LIN {X 0,Y 406.191,Z 782.909,A -85,B 0,C 180,E1 -7084.724,E2 -7084.724} C_VEL
LIN {X 0,Y 404.548,Z 789.361,A -85,B 0,C 180,E1 -7085.289,E2 -7085.289} C_VEL
LIN {X 0,Y 396.99,Z 805.186,A -85,B 0,C 180,E1 -7086.699,E2 -7086.699} C_VEL
LIN {X 0,Y 395.215,Z 810.941,A -85,B 0,C 180,E1 -7087.406,E2 -7087.406} C_VEL
LIN {X 0,Y 393.105,Z 824.076,A -85,B 0,C 180,E1 -7089.452,E2 -7089.452} C_VEL
LIN {X 0,Y 391.138,Z 835.792,A -85,B 0,C 180,E1 -7091.674,E2 -7091.674} C_VEL
LIN {X 0,Y 389.418,Z 846.025,A -85,B 0,C 180,E1 -7094.054,E2 -7094.054} C_VEL
LIN {X 0,Y 388.003,Z 854.789,A -85,B 0,C 180,E1 -7096.59,E2 -7096.59} C_VEL
LIN {X 0,Y 386.881,Z 862.038,A -85,B 0,C 180,E1 -7099.276,E2 -7099.276} C_VEL
LIN {X 0,Y 386.108,Z 867.692,A -85,B 0,C 180,E1 -7102.112,E2 -7102.112} C_VEL
LIN {X 0,Y 385.668,Z 871.52,A -85,B 0,C 180,E1 -7104.943,E2 -7104.943} C_VEL
LIN {X 0,Y 385.436,Z 873.652,A -85,B 0,C 180,E1 -7107.77,E2 -7107.77} C_VEL
LIN {X 0,Y 385.386,Z 874.148,A -85,B 0,C 180,E1 -7110.595,E2 -7110.595} C_VEL
LIN {X 0,Y 385.508,Z 872.915,A -85,B 0,C 180,E1 -7113.569,E2 -7113.569} C_VEL
LIN {X 0,Y 385.826,Z 870.044,A -85,B 0,C 180,E1 -7116.398,E2 -7116.398} C_VEL
LIN {X 0,Y 386.363,Z 865.702,A -85,B 0,C 180,E1 -7119.083,E2 -7119.083} C_VEL
LIN {X 0,Y 387.229,Z 859.657,A -85,B 0,C 180,E1 -7121.771,E2 -7121.771} C_VEL
LIN {X 0,Y 388.409,Z 852.203,A -85,B 0,C 180,E1 -7124.308,E2 -7124.308} C_VEL
LIN {X 0,Y 389.961,Z 842.815,A -85,B 0,C 180,E1 -7126.842,E2 -7126.842} C_VEL
LIN {X 0,Y 391.848,Z 831.752,A -85,B 0,C 180,E1 -7129.245,E2 -7129.245} C_VEL
LIN {X 0,Y 393.914,Z 819.324,A -85,B 0,C 180,E1 -7131.439,E2 -7131.439} C_VEL
LIN {X 0,Y 396.073,Z 805.549,A -85,B 0,C 180,E1 -7133.429,E2 -7133.429} C_VEL
LIN {X 0,Y 398.217,Z 790.671,A -85,B 0,C 180,E1 -7135.188,E2 -7135.188} C_VEL
LIN {X 0,Y 400.199,Z 774.726,A -85,B 0,C 180,E1 -7136.726,E2 -7136.726} C_VEL
LIN {X 0,Y 401.902,Z 758.677,A -85,B 0,C 180,E1 -7137.971,E2 -7137.971} C_VEL
LIN {X 0,Y 403.321,Z 741.862,A -85,B 0,C 180,E1 -7139.001,E2 -7139.001} C_VEL
LIN {X 0,Y 404.378,Z 723.64,A -85,B 0,C 180,E1 -7139.842,E2 -7139.842} C_VEL
LIN {X 0,Y 404.994,Z 704.322,A -85,B 0,C 180,E1 -7140.452,E2 -7140.452} C_VEL
LIN {X 0,Y 406.775,Z 627.656,A -85,B 0,C 180,E1 -7141.895,E2 -7141.895} C_VEL
LIN {X 0,Y 409.987,Z 503.447,A -85,B 0,C 180,E1 -7144.179,E2 -7144.179} C_VEL
LIN {X 0,Y 409.147,Z 496.442,A -85,B 0,C 180,E1 -7144.454,E2 -7144.454} C_VEL
LIN {X 0,Y 410.584,Z 460.846,A -85,B 0,C 180,E1 -7147.153,E2 -7147.153} C_VEL
LIN {X 0,Y 411.5,Z 441.452,A -85,B 0,C 180,E1 -7148.742,E2 -7148.742} C_VEL
LIN {X 0,Y 404.352,Z 422.499,A -85,B 0,C 180,E1 -7151.318,E2 -7151.318} C_VEL
LIN {X 0,Y 399.341,Z 410.865,A -85,B 0,C 180,E1 -7153.021,E2 -7153.021} C_VEL
LIN {X 0,Y 398.731,Z 410.597,A -85,B 0,C 180,E1 -7153.158,E2 -7153.158} C_VEL
LIN {X 0,Y 405.761,Z 426.901,A -85,B 0,C 180,E1 -7156.118,E2 -7156.118} C_VEL
LIN {X 0,Y 412.622,Z 444.419,A -85,B 0,C 180,E1 -7159.01,E2 -7159.01} C_VEL
LIN {X 0,Y 414.278,Z 448.803,A -85,B 0,C 180,E1 -7159.7,E2 -7159.7} C_VEL
LIN {X 0,Y 409.876,Z 489.947,A -85,B 0,C 180,E1 -7163.645,E2 -7163.645} C_VEL
LIN {X 0,Y 405.47,Z 533.935,A -85,B 0,C 180,E1 -7167.816,E2 -7167.816} C_VEL
LIN {X 0,Y 401.479,Z 578.727,A -85,B 0,C 180,E1 -7172.001,E2 -7172.001} C_VEL
LIN {X 0,Y 399.443,Z 605.362,A -85,B 0,C 180,E1 -7174.432,E2 -7174.432} C_VEL
LIN {X 0,Y 400.173,Z 614.62,A -85,B 0,C 180,E1 -7174.744,E2 -7174.744} C_VEL
LIN {X 0,Y 394.659,Z 751.079,A -85,B 0,C 180,E1 -7178.197,E2 -7178.197} C_VEL
LIN {X 0,Y 394.114,Z 767.215,A -85,B 0,C 180,E1 -7178.833,E2 -7178.833} C_VEL
LIN {X 0,Y 393.253,Z 783.894,A -85,B 0,C 180,E1 -7179.77,E2 -7179.77} C_VEL
LIN {X 0,Y 392.264,Z 798.711,A -85,B 0,C 180,E1 -7180.88,E2 -7180.88} C_VEL
LIN {X 0,Y 391.095,Z 813.488,A -85,B 0,C 180,E1 -7182.288,E2 -7182.288} C_VEL
LIN {X 0,Y 389.952,Z 826.524,A -85,B 0,C 180,E1 -7183.847,E2 -7183.847} C_VEL
LIN {X 0,Y 388.794,Z 839.087,A -85,B 0,C 180,E1 -7185.706,E2 -7185.706} C_VEL
LIN {X 0,Y 387.824,Z 849.553,A -85,B 0,C 180,E1 -7187.644,E2 -7187.644} C_VEL
LIN {X 0,Y 386.992,Z 859.155,A -85,B 0,C 180,E1 -7189.862,E2 -7189.862} C_VEL
LIN {X 0,Y 386.402,Z 866.658,A -85,B 0,C 180,E1 -7192.117,E2 -7192.117} C_VEL
LIN {X 0,Y 386.036,Z 872.623,A -85,B 0,C 180,E1 -7194.5,E2 -7194.5} C_VEL
LIN {X 0,Y 385.892,Z 876.86,A -85,B 0,C 180,E1 -7197.029,E2 -7197.029} C_VEL
LIN {X 0,Y 385.925,Z 879.099,A -85,B 0,C 180,E1 -7199.406,E2 -7199.406} C_VEL
LIN {X 0,Y 386.147,Z 879.624,A -85,B 0,C 180,E1 -7201.929,E2 -7201.929} C_VEL
LIN {X 0,Y 386.531,Z 878.409,A -85,B 0,C 180,E1 -7204.302,E2 -7204.302} C_VEL
LIN {X 0,Y 387.2,Z 875.274,A -85,B 0,C 180,E1 -7206.822,E2 -7206.822} C_VEL
LIN {X 0,Y 388.11,Z 870.426,A -85,B 0,C 180,E1 -7209.191,E2 -7209.191} C_VEL
LIN {X 0,Y 389.28,Z 864.13,A -85,B 0,C 180,E1 -7211.406,E2 -7211.406} C_VEL
LIN {X 0,Y 390.71,Z 855.743,A -85,B 0,C 180,E1 -7213.617,E2 -7213.617} C_VEL
LIN {X 0,Y 392.242,Z 846.555,A -85,B 0,C 180,E1 -7215.524,E2 -7215.524} C_VEL
LIN {X 0,Y 394.103,Z 834.538,A -85,B 0,C 180,E1 -7217.496,E2 -7217.496} C_VEL
LIN {X 0,Y 395.961,Z 821.007,A -85,B 0,C 180,E1 -7219.24,E2 -7219.24} C_VEL
LIN {X 0,Y 397.722,Z 805.897,A -85,B 0,C 180,E1 -7220.76,E2 -7220.76} C_VEL
LIN {X 0,Y 399.098,Z 790.974,A -85,B 0,C 180,E1 -7221.918,E2 -7221.918} C_VEL
LIN {X 0,Y 400.201,Z 775.813,A -85,B 0,C 180,E1 -7222.822,E2 -7222.822} C_VEL
LIN {X 0,Y 402.733,Z 747.163,A -85,B 0,C 180,E1 -7224.182,E2 -7224.182} C_VEL
LIN {X 0,Y 414.664,Z 670.102,A -85,B 0,C 180,E1 -7227.461,E2 -7227.461} C_VEL
LIN {X 0,Y 419.144,Z 642.978,A -85,B 0,C 180,E1 -7228.495,E2 -7228.495} C_VEL
LIN {X 0,Y 425.346,Z 629.291,A -85,B 0,C 180,E1 -7229.425,E2 -7229.425} C_VEL
LIN {X 0,Y 433.429,Z 606.324,A -85,B 0,C 180,E1 -7232.2,E2 -7232.2} C_VEL
LIN {X 0,Y 442.63,Z 586.799,A -85,B 0,C 180,E1 -7234.697,E2 -7234.697} C_VEL
LIN {X 0,Y 451.342,Z 572.774,A -85,B 0,C 180,E1 -7236.588,E2 -7236.588} C_VEL
LIN {X 0,Y 449.087,Z 580.004,A -85,B 0,C 180,E1 -7238.239,E2 -7238.239} C_VEL
LIN {X 0,Y 449.02,Z 587.826,A -85,B 0,C 180,E1 -7240.003,E2 -7240.003} C_VEL
LIN {X 0,Y 451.418,Z 596.121,A -85,B 0,C 180,E1 -7241.812,E2 -7241.812} C_VEL
LIN {X 0,Y 456.495,Z 604.734,A -85,B 0,C 180,E1 -7243.625,E2 -7243.625} C_VEL
LIN {X 0,Y 459.602,Z 608.735,A -85,B 0,C 180,E1 -7244.43,E2 -7244.43} C_VEL
LIN {X 0,Y 448.07,Z 630.938,A -85,B 0,C 180,E1 -7244.977,E2 -7244.977} C_VEL
LIN {X 0,Y 439.647,Z 649.717,A -85,B 0,C 180,E1 -7245.626,E2 -7245.626} C_VEL
LIN {X 0,Y 428.488,Z 674.951,A -85,B 0,C 180,E1 -7246.527,E2 -7246.527} C_VEL
LIN {X 0,Y 420.017,Z 698.201,A -85,B 0,C 180,E1 -7247.552,E2 -7247.552} C_VEL
LIN {X 0,Y 416.651,Z 725.416,A -85,B 0,C 180,E1 -7248.015,E2 -7248.015} C_VEL
LIN {X 0,Y 414.363,Z 753.273,A -85,B 0,C 180,E1 -7248.807,E2 -7248.807} C_VEL
LIN {X 0,Y 411.564,Z 778.053,A -85,B 0,C 180,E1 -7249.742,E2 -7249.742} C_VEL
LIN {X 0,Y 408.571,Z 802.272,A -85,B 0,C 180,E1 -7250.938,E2 -7250.938} C_VEL
LIN {X 0,Y 405.472,Z 825.859,A -85,B 0,C 180,E1 -7252.387,E2 -7252.387} C_VEL
LIN {X 0,Y 402.205,Z 849.287,A -85,B 0,C 180,E1 -7254.157,E2 -7254.157} C_VEL
LIN {X 0,Y 399.157,Z 870.873,A -85,B 0,C 180,E1 -7256.105,E2 -7256.105} C_VEL
LIN {X 0,Y 396.34,Z 890.303,A -85,B 0,C 180,E1 -7258.18,E2 -7258.18} C_VEL
LIN {X 0,Y 393.688,Z 908.695,A -85,B 0,C 180,E1 -7260.481,E2 -7260.481} C_VEL
LIN {X 0,Y 391.243,Z 925.999,A -85,B 0,C 180,E1 -7263.023,E2 -7263.023} C_VEL
LIN {X 0,Y 389.144,Z 941.582,A -85,B 0,C 180,E1 -7265.726,E2 -7265.726} C_VEL
LIN {X 0,Y 387.348,Z 956.066,A -85,B 0,C 180,E1 -7268.723,E2 -7268.723} C_VEL
LIN {X 0,Y 386.035,Z 968.119,A -85,B 0,C 180,E1 -7271.735,E2 -7271.735} C_VEL
LIN {X 0,Y 385.139,Z 978.117,A -85,B 0,C 180,E1 -7274.799,E2 -7274.799} C_VEL
LIN {X 0,Y 384.644,Z 985.702,A -85,B 0,C 180,E1 -7277.692,E2 -7277.692} C_VEL
LIN {X 0,Y 384.372,Z 991.86,A -85,B 0,C 180,E1 -7280.718,E2 -7280.718} C_VEL
LIN {X 0,Y 384.304,Z 996.2,A -85,B 0,C 180,E1 -7283.726,E2 -7283.726} C_VEL
LIN {X 0,Y 384.277,Z 998.794,A -85,B 0,C 180,E1 -7286.569,E2 -7286.569} C_VEL
LIN {X 0,Y 384.268,Z 999.915,A -85,B 0,C 180,E1 -7289.403,E2 -7289.403} C_VEL
LIN {X 0,Y 384.257,Z 999.607,A -85,B 0,C 180,E1 -7292.318,E2 -7292.318} C_VEL
LIN {X 0,Y 384.23,Z 997.595,A -85,B 0,C 180,E1 -7295.375,E2 -7295.375} C_VEL
LIN {X 0,Y 384.269,Z 994.042,A -85,B 0,C 180,E1 -7298.378,E2 -7298.378} C_VEL
LIN {X 0,Y 384.465,Z 988.521,A -85,B 0,C 180,E1 -7301.551,E2 -7301.551} C_VEL
LIN {X 0,Y 384.938,Z 981.054,A -85,B 0,C 180,E1 -7304.747,E2 -7304.747} C_VEL
LIN {X 0,Y 385.742,Z 972.533,A -85,B 0,C 180,E1 -7307.654,E2 -7307.654} C_VEL
LIN {X 0,Y 386.969,Z 962.18,A -85,B 0,C 180,E1 -7310.573,E2 -7310.573} C_VEL
LIN {X 0,Y 388.686,Z 949.733,A -85,B 0,C 180,E1 -7313.498,E2 -7313.498} C_VEL
LIN {X 0,Y 390.985,Z 934.899,A -85,B 0,C 180,E1 -7316.421,E2 -7316.421} C_VEL
LIN {X 0,Y 393.76,Z 918.176,A -85,B 0,C 180,E1 -7319.178,E2 -7319.178} C_VEL
LIN {X 0,Y 396.865,Z 900.084,A -85,B 0,C 180,E1 -7321.688,E2 -7321.688} C_VEL
LIN {X 0,Y 399.796,Z 882.701,A -85,B 0,C 180,E1 -7323.724,E2 -7323.724} C_VEL
LIN {X 0,Y 403.015,Z 863.268,A -85,B 0,C 180,E1 -7325.663,E2 -7325.663} C_VEL
LIN {X 0,Y 406.074,Z 843.952,A -85,B 0,C 180,E1 -7327.28,E2 -7327.28} C_VEL
LIN {X 0,Y 409.131,Z 823.037,A -85,B 0,C 180,E1 -7328.728,E2 -7328.728} C_VEL
LIN {X 0,Y 411.966,Z 801.587,A -85,B 0,C 180,E1 -7329.937,E2 -7329.937} C_VEL
LIN {X 0,Y 414.421,Z 780.045,A -85,B 0,C 180,E1 -7330.888,E2 -7330.888} C_VEL
LIN {X 0,Y 416.514,Z 757.64,A -85,B 0,C 180,E1 -7331.614,E2 -7331.614} C_VEL
LIN {X 0,Y 418.138,Z 728.034,A -85,B 0,C 180,E1 -7332.297,E2 -7332.297} C_VEL
LIN {X 0,Y 419.757,Z 710.11,A -85,B 0,C 180,E1 -7332.606,E2 -7332.606} C_VEL
LIN {X 0,Y 425.98,Z 692.528,A -85,B 0,C 180,E1 -7333.45,E2 -7333.45} C_VEL
LIN {X 0,Y 433.679,Z 672.802,A -85,B 0,C 180,E1 -7334.312,E2 -7334.312} C_VEL
LIN {X 0,Y 443.478,Z 651.646,A -85,B 0,C 180,E1 -7335.067,E2 -7335.067} C_VEL
LIN {X 0,Y 452.464,Z 632.249,A -85,B 0,C 180,E1 -7335.723,E2 -7335.723} C_VEL
LIN {X 0,Y 463.366,Z 611.6,A -85,B 0,C 180,E1 -7336.255,E2 -7336.255} C_VEL
LIN {X 0,Y 454.291,Z 599.638,A -85,B 0,C 180,E1 -7338.174,E2 -7338.174} C_VEL
LIN {X 0,Y 447.091,Z 586.383,A -85,B 0,C 180,E1 -7340.091,E2 -7340.091} C_VEL
LIN {X 0,Y 441.688,Z 571.997,A -85,B 0,C 180,E1 -7341.995,E2 -7341.995} C_VEL
LIN {X 0,Y 438.002,Z 555.946,A -85,B 0,C 180,E1 -7343.918,E2 -7343.918} C_VEL
LIN {X 0,Y 436.131,Z 538.265,A -85,B 0,C 180,E1 -7345.828,E2 -7345.828} C_VEL
LIN {X 0,Y 436.157,Z 518.452,A -85,B 0,C 180,E1 -7347.769,E2 -7347.769} C_VEL
LIN {X 0,Y 438.293,Z 495.895,A -85,B 0,C 180,E1 -7349.725,E2 -7349.725} C_VEL
LIN {X 0,Y 440.506,Z 480.25,A -85,B 0,C 180,E1 -7351.014,E2 -7351.014} C_VEL
LIN {X 0,Y 431.282,Z 462.851,A -85,B 0,C 180,E1 -7354.4,E2 -7354.4} C_VEL
LIN {X 0,Y 422.428,Z 446.642,A -85,B 0,C 180,E1 -7357.893,E2 -7357.893} C_VEL
LIN {X 0,Y 414.929,Z 433.34,A -85,B 0,C 180,E1 -7361.016,E2 -7361.016} C_VEL
LIN {X 0,Y 406.659,Z 418.792,A -85,B 0,C 180,E1 -7364.747,E2 -7364.747} C_VEL
LIN {X 0,Y 400.297,Z 408.182,A -85,B 0,C 180,E1 -7367.743,E2 -7367.743} C_VEL
LIN {X 0,Y 397.265,Z 403.054,A -85,B 0,C 180,E1 -7369.267,E2 -7369.267} C_VEL
LIN {X 0,Y 394.273,Z 397.969,A -85,B 0,C 180,E1 -7370.807,E2 -7370.807} C_VEL
LIN {X 0,Y 392.155,Z 394.36,A -85,B 0,C 180,E1 -7371.939,E2 -7371.939} C_VEL
LIN {X 0,Y 391.365,Z 392.977,A -85,B 0,C 180,E1 -7372.366,E2 -7372.366} C_VEL
LIN {X 0,Y 389.215,Z 389.622,A -85,B 0,C 180,E1 -7373.51,E2 -7373.51} C_VEL
LIN {X 0,Y 388.631,Z 388.038,A -85,B 0,C 180,E1 -7373.945,E2 -7373.945} C_VEL
LIN {X 0,Y 386.273,Z 385.055,A -85,B 0,C 180,E1 -7375.1,E2 -7375.1} C_VEL
LIN {X 0,Y 385.581,Z 382.706,A -85,B 0,C 180,E1 -7375.762,E2 -7375.762} C_VEL
LIN {X 0,Y 385.627,Z 382.705,A -85,B 0,C 180,E1 -7379.852,E2 -7379.852} C_VEL
LIN {X 0,Y 385.585,Z 382.712,A -85,B 0,C 180,E1 -7384.015,E2 -7384.015} C_VEL
LIN {X 0,Y 385.623,Z 382.701,A -85,B 0,C 180,E1 -7387.921,E2 -7387.921} C_VEL
LIN {X 0,Y 385.595,Z 382.705,A -85,B 0,C 180,E1 -7392.125,E2 -7392.125} C_VEL
LIN {X 0,Y 385.621,Z 382.697,A -85,B 0,C 180,E1 -7395.953,E2 -7395.953} C_VEL
LIN {X 0,Y 385.607,Z 382.702,A -85,B 0,C 180,E1 -7400.175,E2 -7400.175} C_VEL
LIN {X 0,Y 385.617,Z 382.696,A -85,B 0,C 180,E1 -7404.121,E2 -7404.121} C_VEL
LIN {X 0,Y 385.616,Z 382.694,A -85,B 0,C 180,E1 -7408.327,E2 -7408.327} C_VEL
LIN {X 0,Y 385.616,Z 382.693,A -85,B 0,C 180,E1 -7412.11,E2 -7412.11} C_VEL
LIN {X 0,Y 385.62,Z 382.653,A -85,B 0,C 180,E1 -7416.057,E2 -7416.057} C_VEL
LIN {X 0,Y 385.596,Z 382.702,A -85,B 0,C 180,E1 -7420.022,E2 -7420.022} C_VEL
LIN {X 0,Y 385.636,Z 382.835,A -85,B 0,C 180,E1 -7422.588,E2 -7422.588} C_VEL
LIN {X 0,Y 386.754,Z 385.913,A -85,B 0,C 180,E1 -7423.041,E2 -7423.041} C_VEL
LIN {X 0,Y 388.166,Z 388.118,A -85,B 0,C 180,E1 -7423.453,E2 -7423.453} C_VEL
LIN {X 0,Y 396.059,Z 403.776,A -85,B 0,C 180,E1 -7426.013,E2 -7426.013} C_VEL
LIN {X 0,Y 404.031,Z 421.706,A -85,B 0,C 180,E1 -7428.684,E2 -7428.684} C_VEL
LIN {X 0,Y 410.869,Z 439.77,A -85,B 0,C 180,E1 -7431.145,E2 -7431.145} C_VEL
LIN {X 0,Y 411.575,Z 442.452,A -85,B 0,C 180,E1 -7431.468,E2 -7431.468} C_VEL
LIN {X 0,Y 409.531,Z 482.811,A -85,B 0,C 180,E1 -7434.646,E2 -7434.646} C_VEL
LIN {X 0,Y 409.192,Z 497.98,A -85,B 0,C 180,E1 -7435.727,E2 -7435.727} C_VEL
LIN {X 0,Y 410.063,Z 506.076,A -85,B 0,C 180,E1 -7435.984,E2 -7435.984} C_VEL
LIN {X 0,Y 404.983,Z 703.514,A -85,B 0,C 180,E1 -7439.625,E2 -7439.625} C_VEL
LIN {X 0,Y 404.404,Z 722.407,A -85,B 0,C 180,E1 -7440.207,E2 -7440.207} C_VEL
LIN {X 0,Y 403.357,Z 740.984,A -85,B 0,C 180,E1 -7441.05,E2 -7441.05} C_VEL
LIN {X 0,Y 401.891,Z 758.5,A -85,B 0,C 180,E1 -7442.114,E2 -7442.114} C_VEL
LIN {X 0,Y 400.17,Z 774.763,A -85,B 0,C 180,E1 -7443.375,E2 -7443.375} C_VEL
LIN {X 0,Y 398.215,Z 790.511,A -85,B 0,C 180,E1 -7444.892,E2 -7444.892} C_VEL
LIN {X 0,Y 396.135,Z 804.974,A -85,B 0,C 180,E1 -7446.595,E2 -7446.595} C_VEL
LIN {X 0,Y 395.215,Z 810.941,A -85,B 0,C 180,E1 -7447.406,E2 -7447.406} C_VEL
LIN {X 0,Y 393.457,Z 816.543,A -85,B 0,C 180,E1 -7448.146,E2 -7448.146} C_VEL
LIN {X 0,Y 386.123,Z 829.485,A -85,B 0,C 180,E1 -7449.887,E2 -7449.887} C_VEL
LIN {X 0,Y 384.132,Z 834.334,A -85,B 0,C 180,E1 -7450.739,E2 -7450.739} C_VEL
LIN {X 0,Y 383.993,Z 834.979,A -85,B 0,C 180,E1 -7450.871,E2 -7450.871} C_VEL
LIN {X 0,Y 382.104,Z 845.532,A -85,B 0,C 180,E1 -7453.281,E2 -7453.281} C_VEL
LIN {X 0,Y 380.528,Z 854.61,A -85,B 0,C 180,E1 -7455.856,E2 -7455.856} C_VEL
LIN {X 0,Y 379.265,Z 862.196,A -85,B 0,C 180,E1 -7458.597,E2 -7458.597} C_VEL
LIN {X 0,Y 378.407,Z 867.917,A -85,B 0,C 180,E1 -7461.338,E2 -7461.338} C_VEL
LIN {X 0,Y 377.865,Z 872.141,A -85,B 0,C 180,E1 -7464.23,E2 -7464.23} C_VEL
LIN {X 0,Y 377.578,Z 874.636,A -85,B 0,C 180,E1 -7467.116,E2 -7467.116} C_VEL
LIN {X 0,Y 377.49,Z 875.482,A -85,B 0,C 180,E1 -7470,E2 -7470} C_VEL
LIN {X 0,Y 377.576,Z 874.7,A -85,B 0,C 180,E1 -7472.884,E2 -7472.884} C_VEL
LIN {X 0,Y 377.857,Z 872.264,A -85,B 0,C 180,E1 -7475.771,E2 -7475.771} C_VEL
LIN {X 0,Y 378.389,Z 868.093,A -85,B 0,C 180,E1 -7478.663,E2 -7478.663} C_VEL
LIN {X 0,Y 379.236,Z 862.432,A -85,B 0,C 180,E1 -7481.405,E2 -7481.405} C_VEL
LIN {X 0,Y 380.41,Z 855.395,A -85,B 0,C 180,E1 -7483.994,E2 -7483.994} C_VEL
LIN {X 0,Y 381.954,Z 846.469,A -85,B 0,C 180,E1 -7486.579,E2 -7486.579} C_VEL
LIN {X 0,Y 383.815,Z 836.05,A -85,B 0,C 180,E1 -7489.004,E2 -7489.004} C_VEL
LIN {X 0,Y 385.927,Z 824.123,A -85,B 0,C 180,E1 -7491.267,E2 -7491.267} C_VEL
LIN {X 0,Y 388.207,Z 810.597,A -85,B 0,C 180,E1 -7493.369,E2 -7493.369} C_VEL
LIN {X 0,Y 390.399,Z 796.548,A -85,B 0,C 180,E1 -7495.16,E2 -7495.16} C_VEL
LIN {X 0,Y 392.545,Z 780.881,A -85,B 0,C 180,E1 -7496.798,E2 -7496.798} C_VEL
LIN {X 0,Y 394.406,Z 765.058,A -85,B 0,C 180,E1 -7498.134,E2 -7498.134} C_VEL
LIN {X 0,Y 395.992,Z 748.492,A -85,B 0,C 180,E1 -7499.248,E2 -7499.248} C_VEL
LIN {X 0,Y 397.246,Z 730.538,A -85,B 0,C 180,E1 -7500.173,E2 -7500.173} C_VEL
LIN {X 0,Y 398.021,Z 712.038,A -85,B 0,C 180,E1 -7500.855,E2 -7500.855} C_VEL
LIN {X 0,Y 398.446,Z 688.282,A -85,B 0,C 180,E1 -7501.392,E2 -7501.392} C_VEL
LIN {X 0,Y 403.431,Z 504.677,A -85,B 0,C 180,E1 -7504.811,E2 -7504.811} C_VEL
LIN {X 0,Y 402.608,Z 497.605,A -85,B 0,C 180,E1 -7505.095,E2 -7505.095} C_VEL
LIN {X 0,Y 404.187,Z 460.96,A -85,B 0,C 180,E1 -7507.895,E2 -7507.895} C_VEL
LIN {X 0,Y 405.077,Z 445.128,A -85,B 0,C 180,E1 -7509.19,E2 -7509.19} C_VEL
LIN {X 0,Y 397.875,Z 426.006,A -85,B 0,C 180,E1 -7511.831,E2 -7511.831} C_VEL
LIN {X 0,Y 394.282,Z 417.655,A -85,B 0,C 180,E1 -7513.085,E2 -7513.085} C_VEL
LIN {X 0,Y 393.596,Z 417.375,A -85,B 0,C 180,E1 -7513.238,E2 -7513.238} C_VEL
LIN {X 0,Y 400.975,Z 434.884,A -85,B 0,C 180,E1 -7516.418,E2 -7516.418} C_VEL
LIN {X 0,Y 407.594,Z 452.337,A -85,B 0,C 180,E1 -7519.268,E2 -7519.268} C_VEL
LIN {X 0,Y 402.837,Z 494.236,A -85,B 0,C 180,E1 -7523.34,E2 -7523.34} C_VEL
LIN {X 0,Y 398.322,Z 537.838,A -85,B 0,C 180,E1 -7527.508,E2 -7527.508} C_VEL
LIN {X 0,Y 394.228,Z 582.079,A -85,B 0,C 180,E1 -7531.687,E2 -7531.687} C_VEL
LIN {X 0,Y 392.309,Z 606.257,A -85,B 0,C 180,E1 -7533.915,E2 -7533.915} C_VEL
LIN {X 0,Y 393.003,Z 615.661,A -85,B 0,C 180,E1 -7534.242,E2 -7534.242} C_VEL
LIN {X 0,Y 387.169,Z 751.411,A -85,B 0,C 180,E1 -7537.788,E2 -7537.788} C_VEL
LIN {X 0,Y 386.586,Z 768.044,A -85,B 0,C 180,E1 -7538.452,E2 -7538.452} C_VEL
LIN {X 0,Y 385.663,Z 785.126,A -85,B 0,C 180,E1 -7539.433,E2 -7539.433} C_VEL
LIN {X 0,Y 384.635,Z 799.902,A -85,B 0,C 180,E1 -7540.565,E2 -7540.565} C_VEL
LIN {X 0,Y 383.418,Z 814.664,A -85,B 0,C 180,E1 -7541.999,E2 -7541.999} C_VEL
LIN {X 0,Y 382.229,Z 827.709,A -85,B 0,C 180,E1 -7543.589,E2 -7543.589} C_VEL
LIN {X 0,Y 381.064,Z 839.826,A -85,B 0,C 180,E1 -7545.41,E2 -7545.41} C_VEL
LIN {X 0,Y 380.047,Z 850.428,A -85,B 0,C 180,E1 -7547.387,E2 -7547.387} C_VEL
LIN {X 0,Y 379.162,Z 860.207,A -85,B 0,C 180,E1 -7549.67,E2 -7549.67} C_VEL
LIN {X 0,Y 378.545,Z 867.747,A -85,B 0,C 180,E1 -7551.952,E2 -7551.952} C_VEL
LIN {X 0,Y 378.158,Z 873.804,A -85,B 0,C 180,E1 -7554.385,E2 -7554.385} C_VEL
LIN {X 0,Y 378.002,Z 878.125,A -85,B 0,C 180,E1 -7556.967,E2 -7556.967} C_VEL
LIN {X 0,Y 378.045,Z 880.477,A -85,B 0,C 180,E1 -7559.393,E2 -7559.393} C_VEL
LIN {X 0,Y 378.287,Z 881.092,A -85,B 0,C 180,E1 -7561.969,E2 -7561.969} C_VEL
LIN {X 0,Y 378.708,Z 879.98,A -85,B 0,C 180,E1 -7564.391,E2 -7564.391} C_VEL
LIN {X 0,Y 379.434,Z 876.956,A -85,B 0,C 180,E1 -7566.962,E2 -7566.962} C_VEL
LIN {X 0,Y 380.416,Z 872.225,A -85,B 0,C 180,E1 -7569.378,E2 -7569.378} C_VEL
LIN {X 0,Y 381.673,Z 866.062,A -85,B 0,C 180,E1 -7571.637,E2 -7571.637} C_VEL
LIN {X 0,Y 383.209,Z 857.848,A -85,B 0,C 180,E1 -7573.889,E2 -7573.889} C_VEL
LIN {X 0,Y 384.979,Z 848.055,A -85,B 0,C 180,E1 -7575.979,E2 -7575.979} C_VEL
LIN {X 0,Y 386.748,Z 837.593,A -85,B 0,C 180,E1 -7577.762,E2 -7577.762} C_VEL
LIN {X 0,Y 388.724,Z 824.551,A -85,B 0,C 180,E1 -7579.534,E2 -7579.534} C_VEL
LIN {X 0,Y 390.417,Z 811.666,A -85,B 0,C 180,E1 -7580.932,E2 -7580.932} C_VEL
LIN {X 0,Y 392.028,Z 797.363,A -85,B 0,C 180,E1 -7582.177,E2 -7582.177} C_VEL
LIN {X 0,Y 393.532,Z 780.194,A -85,B 0,C 180,E1 -7583.31,E2 -7583.31} C_VEL
LIN {X 0,Y 396.217,Z 752.594,A -85,B 0,C 180,E1 -7584.725,E2 -7584.725} C_VEL
LIN {X 0,Y 405.058,Z 699.54,A -85,B 0,C 180,E1 -7587.171,E2 -7587.171} C_VEL
LIN {X 0,Y 414.422,Z 646.206,A -85,B 0,C 180,E1 -7589.325,E2 -7589.325} C_VEL
LIN {X 0,Y 421.181,Z 631.89,A -85,B 0,C 180,E1 -7590.295,E2 -7590.295} C_VEL
LIN {X 0,Y 429.699,Z 610.164,A -85,B 0,C 180,E1 -7592.989,E2 -7592.989} C_VEL
LIN {X 0,Y 439.07,Z 592.219,A -85,B 0,C 180,E1 -7595.339,E2 -7595.339} C_VEL
LIN {X 0,Y 446.111,Z 581.569,A -85,B 0,C 180,E1 -7596.795,E2 -7596.795} C_VEL
LIN {X 0,Y 444.248,Z 589.049,A -85,B 0,C 180,E1 -7598.567,E2 -7598.567} C_VEL
LIN {X 0,Y 444.604,Z 596.015,A -85,B 0,C 180,E1 -7600.197,E2 -7600.197} C_VEL
LIN {X 0,Y 447.185,Z 603.78,A -85,B 0,C 180,E1 -7601.953,E2 -7601.953} C_VEL
LIN {X 0,Y 452.207,Z 612.173,A -85,B 0,C 180,E1 -7603.741,E2 -7603.741} C_VEL
LIN {X 0,Y 441.401,Z 633.32,A -85,B 0,C 180,E1 -7604.29,E2 -7604.29} C_VEL
LIN {X 0,Y 431.202,Z 655.913,A -85,B 0,C 180,E1 -7605.084,E2 -7605.084} C_VEL
LIN {X 0,Y 422.826,Z 674.76,A -85,B 0,C 180,E1 -7605.766,E2 -7605.766} C_VEL
LIN {X 0,Y 414.938,Z 695.886,A -85,B 0,C 180,E1 -7606.703,E2 -7606.703} C_VEL
LIN {X 0,Y 410.992,Z 725.478,A -85,B 0,C 180,E1 -7607.23,E2 -7607.23} C_VEL
LIN {X 0,Y 408.277,Z 753.897,A -85,B 0,C 180,E1 -7608.089,E2 -7608.089} C_VEL
LIN {X 0,Y 404.971,Z 779.847,A -85,B 0,C 180,E1 -7609.135,E2 -7609.135} C_VEL
LIN {X 0,Y 401.828,Z 803.028,A -85,B 0,C 180,E1 -7610.339,E2 -7610.339} C_VEL
LIN {X 0,Y 398.546,Z 825.76,A -85,B 0,C 180,E1 -7611.799,E2 -7611.799} C_VEL
LIN {X 0,Y 394.955,Z 849.755,A -85,B 0,C 180,E1 -7613.673,E2 -7613.673} C_VEL
LIN {X 0,Y 391.735,Z 871.035,A -85,B 0,C 180,E1 -7615.661,E2 -7615.661} C_VEL
LIN {X 0,Y 388.511,Z 891.955,A -85,B 0,C 180,E1 -7617.984,E2 -7617.984} C_VEL
LIN {X 0,Y 385.616,Z 910.998,A -85,B 0,C 180,E1 -7620.485,E2 -7620.485} C_VEL
LIN {X 0,Y 383.013,Z 928.646,A -85,B 0,C 180,E1 -7623.225,E2 -7623.225} C_VEL
LIN {X 0,Y 380.817,Z 944.473,A -85,B 0,C 180,E1 -7626.15,E2 -7626.15} C_VEL
LIN {X 0,Y 379.118,Z 958.005,A -85,B 0,C 180,E1 -7629.142,E2 -7629.142} C_VEL
LIN {X 0,Y 377.9,Z 969.213,A -85,B 0,C 180,E1 -7632.126,E2 -7632.126} C_VEL
LIN {X 0,Y 377.124,Z 977.967,A -85,B 0,C 180,E1 -7634.94,E2 -7634.94} C_VEL
LIN {X 0,Y 376.638,Z 985.725,A -85,B 0,C 180,E1 -7638.049,E2 -7638.049} C_VEL
LIN {X 0,Y 376.418,Z 991.323,A -85,B 0,C 180,E1 -7640.983,E2 -7640.983} C_VEL
LIN {X 0,Y 376.364,Z 995.535,A -85,B 0,C 180,E1 -7644.053,E2 -7644.053} C_VEL
LIN {X 0,Y 376.346,Z 998.001,A -85,B 0,C 180,E1 -7647.106,E2 -7647.106} C_VEL
LIN {X 0,Y 376.364,Z 998.887,A -85,B 0,C 180,E1 -7650,E2 -7650} C_VEL
LIN {X 0,Y 376.321,Z 998.188,A -85,B 0,C 180,E1 -7653.046,E2 -7653.046} C_VEL
LIN {X 0,Y 376.295,Z 995.921,A -85,B 0,C 180,E1 -7656.101,E2 -7656.101} C_VEL
LIN {X 0,Y 376.335,Z 991.768,A -85,B 0,C 180,E1 -7659.326,E2 -7659.326} C_VEL
LIN {X 0,Y 376.58,Z 986.069,A -85,B 0,C 180,E1 -7662.419,E2 -7662.419} C_VEL
LIN {X 0,Y 377.136,Z 978.61,A -85,B 0,C 180,E1 -7665.531,E2 -7665.531} C_VEL
LIN {X 0,Y 378.103,Z 969.234,A -85,B 0,C 180,E1 -7668.661,E2 -7668.661} C_VEL
LIN {X 0,Y 379.598,Z 957.724,A -85,B 0,C 180,E1 -7671.801,E2 -7671.801} C_VEL
LIN {X 0,Y 381.707,Z 943.786,A -85,B 0,C 180,E1 -7674.943,E2 -7674.943} C_VEL
LIN {X 0,Y 384.217,Z 928.771,A -85,B 0,C 180,E1 -7677.775,E2 -7677.775} C_VEL
LIN {X 0,Y 387.221,Z 911.662,A -85,B 0,C 180,E1 -7680.49,E2 -7680.49} C_VEL
LIN {X 0,Y 390.526,Z 893.107,A -85,B 0,C 180,E1 -7682.96,E2 -7682.96} C_VEL
LIN {X 0,Y 394.089,Z 872.762,A -85,B 0,C 180,E1 -7685.219,E2 -7685.219} C_VEL
LIN {X 0,Y 397.277,Z 854.026,A -85,B 0,C 180,E1 -7686.978,E2 -7686.978} C_VEL
LIN {X 0,Y 400.496,Z 833.764,A -85,B 0,C 180,E1 -7688.552,E2 -7688.552} C_VEL
LIN {X 0,Y 403.684,Z 811.821,A -85,B 0,C 180,E1 -7689.954,E2 -7689.954} C_VEL
LIN {X 0,Y 406.488,Z 790.339,A -85,B 0,C 180,E1 -7691.052,E2 -7691.052} C_VEL
LIN {X 0,Y 408.873,Z 768.377,A -85,B 0,C 180,E1 -7691.899,E2 -7691.899} C_VEL
LIN {X 0,Y 410.73,Z 745.058,A -85,B 0,C 180,E1 -7692.556,E2 -7692.556} C_VEL
LIN {X 0,Y 412.346,Z 717.41,A -85,B 0,C 180,E1 -7693.123,E2 -7693.123} C_VEL
LIN {X 0,Y 413.31,Z 709.42,A -85,B 0,C 180,E1 -7693.253,E2 -7693.253} C_VEL
LIN {X 0,Y 419.946,Z 691.129,A -85,B 0,C 180,E1 -7694.14,E2 -7694.14} C_VEL
LIN {X 0,Y 427.725,Z 671.48,A -85,B 0,C 180,E1 -7695.001,E2 -7695.001} C_VEL
LIN {X 0,Y 437.589,Z 650.32,A -85,B 0,C 180,E1 -7695.751,E2 -7695.751} C_VEL
LIN {X 0,Y 446.584,Z 631.147,A -85,B 0,C 180,E1 -7696.403,E2 -7696.403} C_VEL
LIN {X 0,Y 455.387,Z 614.404,A -85,B 0,C 180,E1 -7696.859,E2 -7696.859} C_VEL
LIN {X 0,Y 446.589,Z 601.87,A -85,B 0,C 180,E1 -7698.835,E2 -7698.835} C_VEL
LIN {X 0,Y 439.365,Z 587.196,A -85,B 0,C 180,E1 -7700.923,E2 -7700.923} C_VEL
LIN {X 0,Y 434.328,Z 571.934,A -85,B 0,C 180,E1 -7702.905,E2 -7702.905} C_VEL
LIN {X 0,Y 431.131,Z 555.076,A -85,B 0,C 180,E1 -7704.89,E2 -7704.89} C_VEL
LIN {X 0,Y 429.836,Z 535.81,A -85,B 0,C 180,E1 -7706.943,E2 -7706.943} C_VEL
LIN {X 0,Y 430.445,Z 516.396,A -85,B 0,C 180,E1 -7708.803,E2 -7708.803} C_VEL
LIN {X 0,Y 433.343,Z 492.246,A -85,B 0,C 180,E1 -7710.867,E2 -7710.867} C_VEL
LIN {X 0,Y 434.523,Z 484.666,A -85,B 0,C 180,E1 -7711.48,E2 -7711.48} C_VEL
LIN {X 0,Y 425.283,Z 467.065,A -85,B 0,C 180,E1 -7714.964,E2 -7714.964} C_VEL
LIN {X 0,Y 415.59,Z 449.366,A -85,B 0,C 180,E1 -7718.846,E2 -7718.846} C_VEL
LIN {X 0,Y 407.285,Z 434.661,A -85,B 0,C 180,E1 -7722.425,E2 -7722.425} C_VEL
LIN {X 0,Y 400.428,Z 422.96,A -85,B 0,C 180,E1 -7725.541,E2 -7725.541} C_VEL
LIN {X 0,Y 395.639,Z 414.604,A -85,B 0,C 180,E1 -7727.892,E2 -7727.892} C_VEL
LIN {X 0,Y 392.261,Z 409.025,A -85,B 0,C 180,E1 -7729.574,E2 -7729.574} C_VEL
LIN {X 0,Y 389.598,Z 404.339,A -85,B 0,C 180,E1 -7730.994,E2 -7730.994} C_VEL
LIN {X 0,Y 387.104,Z 399.899,A -85,B 0,C 180,E1 -7732.356,E2 -7732.356} C_VEL
LIN {X 0,Y 384.503,Z 395.948,A -85,B 0,C 180,E1 -7733.73,E2 -7733.73} C_VEL
LIN {X 0,Y 383.502,Z 394.067,A -85,B 0,C 180,E1 -7734.315,E2 -7734.315} C_VEL
LIN {X 0,Y 381.15,Z 390.329,A -85,B 0,C 180,E1 -7735.637,E2 -7735.637} C_VEL
LIN {X 0,Y 380.492,Z 388.872,A -85,B 0,C 180,E1 -7736.083,E2 -7736.083} C_VEL
LIN {X 0,Y 378.249,Z 385.848,A -85,B 0,C 180,E1 -7737.273,E2 -7737.273} C_VEL
LIN {X 0,Y 377.669,Z 383.693,A -85,B 0,C 180,E1 -7737.876,E2 -7737.876} C_VEL
LIN {X 0,Y 377.662,Z 383.699,A -85,B 0,C 180,E1 -7741.669,E2 -7741.669} C_VEL
LIN {X 0,Y 377.675,Z 383.693,A -85,B 0,C 180,E1 -7745.927,E2 -7745.927} C_VEL
LIN {X 0,Y 377.662,Z 383.692,A -85,B 0,C 180,E1 -7749.756,E2 -7749.756} C_VEL
LIN {X 0,Y 377.681,Z 383.692,A -85,B 0,C 180,E1 -7753.941,E2 -7753.941} C_VEL
LIN {X 0,Y 377.662,Z 383.687,A -85,B 0,C 180,E1 -7757.886,E2 -7757.886} C_VEL
LIN {X 0,Y 377.692,Z 383.688,A -85,B 0,C 180,E1 -7761.918,E2 -7761.918} C_VEL
LIN {X 0,Y 377.67,Z 383.689,A -85,B 0,C 180,E1 -7765.902,E2 -7765.902} C_VEL
LIN {X 0,Y 377.689,Z 383.689,A -85,B 0,C 180,E1 -7769.848,E2 -7769.848} C_VEL
LIN {X 0,Y 377.681,Z 383.682,A -85,B 0,C 180,E1 -7774.043,E2 -7774.043} C_VEL
LIN {X 0,Y 377.68,Z 383.656,A -85,B 0,C 180,E1 -7778.162,E2 -7778.162} C_VEL
LIN {X 0,Y 377.65,Z 383.714,A -85,B 0,C 180,E1 -7781.411,E2 -7781.411} C_VEL
LIN {X 0,Y 378.829,Z 386.913,A -85,B 0,C 180,E1 -7781.902,E2 -7781.902} C_VEL
LIN {X 0,Y 380.242,Z 388.922,A -85,B 0,C 180,E1 -7782.312,E2 -7782.312} C_VEL
LIN {X 0,Y 388.504,Z 404.998,A -85,B 0,C 180,E1 -7785.052,E2 -7785.052} C_VEL
LIN {X 0,Y 396.6,Z 422.919,A -85,B 0,C 180,E1 -7787.834,E2 -7787.834} C_VEL
LIN {X 0,Y 403.866,Z 441.828,A -85,B 0,C 180,E1 -7790.487,E2 -7790.487} C_VEL
LIN {X 0,Y 405.012,Z 445.847,A -85,B 0,C 180,E1 -7790.986,E2 -7790.986} C_VEL
LIN {X 0,Y 402.889,Z 487.248,A -85,B 0,C 180,E1 -7794.246,E2 -7794.246} C_VEL
LIN {X 0,Y 402.651,Z 499.234,A -85,B 0,C 180,E1 -7795.093,E2 -7795.093} C_VEL
LIN {X 0,Y 403.496,Z 507.223,A -85,B 0,C 180,E1 -7795.352,E2 -7795.352} C_VEL
LIN {X 0,Y 398.159,Z 704.5,A -85,B 0,C 180,E1 -7799.043,E2 -7799.043} C_VEL
LIN {X 0,Y 397.568,Z 723.272,A -85,B 0,C 180,E1 -7799.626,E2 -7799.626} C_VEL
LIN {X 0,Y 396.509,Z 741.461,A -85,B 0,C 180,E1 -7800.456,E2 -7800.456} C_VEL
LIN {X 0,Y 395.028,Z 758.667,A -85,B 0,C 180,E1 -7801.503,E2 -7801.503} C_VEL
LIN {X 0,Y 393.149,Z 775.782,A -85,B 0,C 180,E1 -7802.839,E2 -7802.839} C_VEL
LIN {X 0,Y 391.073,Z 791.766,A -85,B 0,C 180,E1 -7804.401,E2 -7804.401} C_VEL
LIN {X 0,Y 388.914,Z 806.09,A -85,B 0,C 180,E1 -7806.114,E2 -7806.114} C_VEL
LIN {X 0,Y 386.787,Z 819.022,A -85,B 0,C 180,E1 -7807.987,E2 -7807.987} C_VEL
LIN {X 0,Y 384.693,Z 831.085,A -85,B 0,C 180,E1 -7810.094,E2 -7810.094} C_VEL
LIN {X 0,Y 383.993,Z 834.979,A -85,B 0,C 180,E1 -7810.871,E2 -7810.871} C_VEL
LIN {X 0,Y 382.265,Z 839.574,A -85,B 0,C 180,E1 -7811.774,E2 -7811.774} C_VEL
LIN {X 0,Y 375.101,Z 850.112,A -85,B 0,C 180,E1 -7813.91,E2 -7813.91} C_VEL
LIN {X 0,Y 373.247,Z 853.86,A -85,B 0,C 180,E1 -7814.912,E2 -7814.912} C_VEL
LIN {X 0,Y 373.131,Z 854.34,A -85,B 0,C 180,E1 -7815.064,E2 -7815.064} C_VEL
LIN {X 0,Y 371.762,Z 861.952,A -85,B 0,C 180,E1 -7817.733,E2 -7817.733} C_VEL
LIN {X 0,Y 370.751,Z 868.058,A -85,B 0,C 180,E1 -7820.532,E2 -7820.532} C_VEL
LIN {X 0,Y 370.09,Z 872.642,A -85,B 0,C 180,E1 -7823.485,E2 -7823.485} C_VEL
LIN {X 0,Y 369.725,Z 875.48,A -85,B 0,C 180,E1 -7826.434,E2 -7826.434} C_VEL
LIN {X 0,Y 369.591,Z 876.661,A -85,B 0,C 180,E1 -7829.38,E2 -7829.38} C_VEL
LIN {X 0,Y 369.642,Z 876.22,A -85,B 0,C 180,E1 -7832.326,E2 -7832.326} C_VEL
LIN {X 0,Y 369.905,Z 874.144,A -85,B 0,C 180,E1 -7835.274,E2 -7835.274} C_VEL
LIN {X 0,Y 370.413,Z 870.37,A -85,B 0,C 180,E1 -7838.226,E2 -7838.226} C_VEL
LIN {X 0,Y 371.233,Z 865.103,A -85,B 0,C 180,E1 -7841.025,E2 -7841.025} C_VEL
LIN {X 0,Y 372.475,Z 858.039,A -85,B 0,C 180,E1 -7843.823,E2 -7843.823} C_VEL
LIN {X 0,Y 374.047,Z 849.487,A -85,B 0,C 180,E1 -7846.461,E2 -7846.461} C_VEL
LIN {X 0,Y 375.941,Z 839.479,A -85,B 0,C 180,E1 -7848.934,E2 -7848.934} C_VEL
LIN {X 0,Y 378.101,Z 828.012,A -85,B 0,C 180,E1 -7851.241,E2 -7851.241} C_VEL
LIN {X 0,Y 380.424,Z 815.016,A -85,B 0,C 180,E1 -7853.383,E2 -7853.383} C_VEL
LIN {X 0,Y 382.764,Z 800.978,A -85,B 0,C 180,E1 -7855.284,E2 -7855.284} C_VEL
LIN {X 0,Y 384.998,Z 785.991,A -85,B 0,C 180,E1 -7856.949,E2 -7856.949} C_VEL
LIN {X 0,Y 387.005,Z 770.126,A -85,B 0,C 180,E1 -7858.385,E2 -7858.385} C_VEL
LIN {X 0,Y 388.787,Z 753.381,A -85,B 0,C 180,E1 -7859.589,E2 -7859.589} C_VEL
LIN {X 0,Y 390.182,Z 735.48,A -85,B 0,C 180,E1 -7860.584,E2 -7860.584} C_VEL
LIN {X 0,Y 391.112,Z 716.825,A -85,B 0,C 180,E1 -7861.333,E2 -7861.333} C_VEL
LIN {X 0,Y 391.56,Z 695.495,A -85,B 0,C 180,E1 -7861.878,E2 -7861.878} C_VEL
LIN {X 0,Y 396.915,Z 505.823,A -85,B 0,C 180,E1 -7865.466,E2 -7865.466} C_VEL
LIN {X 0,Y 396.12,Z 498.767,A -85,B 0,C 180,E1 -7865.757,E2 -7865.757} C_VEL
LIN {X 0,Y 397.836,Z 461.33,A -85,B 0,C 180,E1 -7868.64,E2 -7868.64} C_VEL
LIN {X 0,Y 398.472,Z 448.18,A -85,B 0,C 180,E1 -7869.739,E2 -7869.739} C_VEL
LIN {X 0,Y 391.329,Z 429.28,A -85,B 0,C 180,E1 -7872.404,E2 -7872.404} C_VEL
LIN {X 0,Y 389.215,Z 424.526,A -85,B 0,C 180,E1 -7873.149,E2 -7873.149} C_VEL
LIN {X 0,Y 388.413,Z 424.145,A -85,B 0,C 180,E1 -7873.311,E2 -7873.311} C_VEL
LIN {X 0,Y 395.651,Z 441.749,A -85,B 0,C 180,E1 -7876.493,E2 -7876.493} C_VEL
LIN {X 0,Y 400.878,Z 455.727,A -85,B 0,C 180,E1 -7878.817,E2 -7878.817} C_VEL
LIN {X 0,Y 396.003,Z 497.209,A -85,B 0,C 180,E1 -7882.882,E2 -7882.882} C_VEL
LIN {X 0,Y 391.262,Z 540.873,A -85,B 0,C 180,E1 -7887.109,E2 -7887.109} C_VEL
LIN {X 0,Y 386.974,Z 585.359,A -85,B 0,C 180,E1 -7891.36,E2 -7891.36} C_VEL
LIN {X 0,Y 385.181,Z 607.074,A -85,B 0,C 180,E1 -7893.383,E2 -7893.383} C_VEL
LIN {X 0,Y 385.858,Z 616.709,A -85,B 0,C 180,E1 -7893.723,E2 -7893.723} C_VEL
LIN {X 0,Y 379.694,Z 751.753,A -85,B 0,C 180,E1 -7897.365,E2 -7897.365} C_VEL
LIN {X 0,Y 379.088,Z 768.643,A -85,B 0,C 180,E1 -7898.045,E2 -7898.045} C_VEL
LIN {X 0,Y 378.16,Z 785.194,A -85,B 0,C 180,E1 -7899.006,E2 -7899.006} C_VEL
LIN {X 0,Y 377.088,Z 800.234,A -85,B 0,C 180,E1 -7900.16,E2 -7900.16} C_VEL
LIN {X 0,Y 375.752,Z 815.839,A -85,B 0,C 180,E1 -7901.7,E2 -7901.7} C_VEL
LIN {X 0,Y 374.511,Z 828.876,A -85,B 0,C 180,E1 -7903.321,E2 -7903.321} C_VEL
LIN {X 0,Y 373.253,Z 841.461,A -85,B 0,C 180,E1 -7905.257,E2 -7905.257} C_VEL
LIN {X 0,Y 372.199,Z 851.982,A -85,B 0,C 180,E1 -7907.274,E2 -7907.274} C_VEL
LIN {X 0,Y 371.284,Z 861.72,A -85,B 0,C 180,E1 -7909.605,E2 -7909.605} C_VEL
LIN {X 0,Y 370.62,Z 869.669,A -85,B 0,C 180,E1 -7912.091,E2 -7912.091} C_VEL
LIN {X 0,Y 370.258,Z 875.276,A -85,B 0,C 180,E1 -7914.421,E2 -7914.421} C_VEL
LIN {X 0,Y 370.112,Z 879.607,A -85,B 0,C 180,E1 -7917.057,E2 -7917.057} C_VEL
LIN {X 0,Y 370.174,Z 881.932,A -85,B 0,C 180,E1 -7919.535,E2 -7919.535} C_VEL
LIN {X 0,Y 370.447,Z 882.561,A -85,B 0,C 180,E1 -7922.165,E2 -7922.165} C_VEL
LIN {X 0,Y 370.927,Z 881.437,A -85,B 0,C 180,E1 -7924.638,E2 -7924.638} C_VEL
LIN {X 0,Y 371.729,Z 878.425,A -85,B 0,C 180,E1 -7927.262,E2 -7927.262} C_VEL
LIN {X 0,Y 372.816,Z 873.708,A -85,B 0,C 180,E1 -7929.727,E2 -7929.727} C_VEL
LIN {X 0,Y 374.192,Z 867.505,A -85,B 0,C 180,E1 -7932.047,E2 -7932.047} C_VEL
LIN {X 0,Y 375.983,Z 858.803,A -85,B 0,C 180,E1 -7934.476,E2 -7934.476} C_VEL
LIN {X 0,Y 377.915,Z 848.856,A -85,B 0,C 180,E1 -7936.603,E2 -7936.603} C_VEL
LIN {X 0,Y 379.928,Z 837.816,A -85,B 0,C 180,E1 -7938.488,E2 -7938.488} C_VEL
LIN {X 0,Y 381.992,Z 825.217,A -85,B 0,C 180,E1 -7940.212,E2 -7940.212} C_VEL
LIN {X 0,Y 384.041,Z 810.787,A -85,B 0,C 180,E1 -7941.777,E2 -7941.777} C_VEL
LIN {X 0,Y 385.888,Z 795.225,A -85,B 0,C 180,E1 -7943.098,E2 -7943.098} C_VEL
LIN {X 0,Y 387.533,Z 777.739,A -85,B 0,C 180,E1 -7944.219,E2 -7944.219} C_VEL
LIN {X 0,Y 390.98,Z 750.474,A -85,B 0,C 180,E1 -7945.687,E2 -7945.687} C_VEL
LIN {X 0,Y 402.375,Z 690.368,A -85,B 0,C 180,E1 -7948.536,E2 -7948.536} C_VEL
LIN {X 0,Y 410.226,Z 649.016,A -85,B 0,C 180,E1 -7950.219,E2 -7950.219} C_VEL
LIN {X 0,Y 417.264,Z 634.812,A -85,B 0,C 180,E1 -7951.17,E2 -7951.17} C_VEL
LIN {X 0,Y 426.674,Z 613.368,A -85,B 0,C 180,E1 -7953.898,E2 -7953.898} C_VEL
LIN {X 0,Y 436.765,Z 596.224,A -85,B 0,C 180,E1 -7956.201,E2 -7956.201} C_VEL
LIN {X 0,Y 440.94,Z 590.4,A -85,B 0,C 180,E1 -7957.043,E2 -7957.043} C_VEL
LIN {X 0,Y 439.58,Z 597.874,A -85,B 0,C 180,E1 -7958.886,E2 -7958.886} C_VEL
LIN {X 0,Y 440.708,Z 605.847,A -85,B 0,C 180,E1 -7960.798,E2 -7960.798} C_VEL
LIN {X 0,Y 444.316,Z 613.779,A -85,B 0,C 180,E1 -7962.636,E2 -7962.636} C_VEL
LIN {X 0,Y 445.245,Z 615.633,A -85,B 0,C 180,E1 -7963.009,E2 -7963.009} C_VEL
LIN {X 0,Y 434.788,Z 636.387,A -85,B 0,C 180,E1 -7963.581,E2 -7963.581} C_VEL
LIN {X 0,Y 426.285,Z 655.024,A -85,B 0,C 180,E1 -7964.249,E2 -7964.249} C_VEL
LIN {X 0,Y 417.417,Z 674.716,A -85,B 0,C 180,E1 -7964.961,E2 -7964.961} C_VEL
LIN {X 0,Y 410.181,Z 693.695,A -85,B 0,C 180,E1 -7965.806,E2 -7965.806} C_VEL
LIN {X 0,Y 405.598,Z 725.619,A -85,B 0,C 180,E1 -7966.399,E2 -7966.399} C_VEL
LIN {X 0,Y 402.572,Z 752.92,A -85,B 0,C 180,E1 -7967.273,E2 -7967.273} C_VEL
LIN {X 0,Y 398.774,Z 779.974,A -85,B 0,C 180,E1 -7968.408,E2 -7968.408} C_VEL
LIN {X 0,Y 395.207,Z 803.68,A -85,B 0,C 180,E1 -7969.699,E2 -7969.699} C_VEL
LIN {X 0,Y 391.369,Z 828.032,A -85,B 0,C 180,E1 -7971.343,E2 -7971.343} C_VEL
LIN {X 0,Y 387.737,Z 850.552,A -85,B 0,C 180,E1 -7973.181,E2 -7973.181} C_VEL
LIN {X 0,Y 384.139,Z 872.534,A -85,B 0,C 180,E1 -7975.335,E2 -7975.335} C_VEL
LIN {X 0,Y 380.894,Z 892.36,A -85,B 0,C 180,E1 -7977.621,E2 -7977.621} C_VEL
LIN {X 0,Y 377.97,Z 910.57,A -85,B 0,C 180,E1 -7980.089,E2 -7980.089} C_VEL
LIN {X 0,Y 375.27,Z 927.942,A -85,B 0,C 180,E1 -7982.86,E2 -7982.86} C_VEL
LIN {X 0,Y 373.022,Z 943.432,A -85,B 0,C 180,E1 -7985.788,E2 -7985.788} C_VEL
LIN {X 0,Y 371.244,Z 956.98,A -85,B 0,C 180,E1 -7988.844,E2 -7988.844} C_VEL
LIN {X 0,Y 369.92,Z 968.778,A -85,B 0,C 180,E1 -7992.067,E2 -7992.067} C_VEL
LIN {X 0,Y 369.112,Z 977.789,A -85,B 0,C 180,E1 -7995.087,E2 -7995.087} C_VEL
LIN {X 0,Y 368.672,Z 985.045,A -85,B 0,C 180,E1 -7998.105,E2 -7998.105} C_VEL
LIN {X 0,Y 368.465,Z 990.804,A -85,B 0,C 180,E1 -8001.259,E2 -8001.259} C_VEL
LIN {X 0,Y 368.434,Z 994.641,A -85,B 0,C 180,E1 -8004.237,E2 -8004.237} C_VEL
LIN {X 0,Y 368.425,Z 997.025,A -85,B 0,C 180,E1 -8007.355,E2 -8007.355} C_VEL
LIN {X 0,Y 368.43,Z 997.752,A -85,B 0,C 180,E1 -8010.311,E2 -8010.311} C_VEL
LIN {X 0,Y 368.392,Z 996.939,A -85,B 0,C 180,E1 -8013.423,E2 -8013.423} C_VEL
LIN {X 0,Y 368.352,Z 994.466,A -85,B 0,C 180,E1 -8016.554,E2 -8016.554} C_VEL
LIN {X 0,Y 368.381,Z 990.39,A -85,B 0,C 180,E1 -8019.687,E2 -8019.687} C_VEL
LIN {X 0,Y 368.681,Z 984.223,A -85,B 0,C 180,E1 -8023.008,E2 -8023.008} C_VEL
LIN {X 0,Y 369.309,Z 976.498,A -85,B 0,C 180,E1 -8026.192,E2 -8026.192} C_VEL
LIN {X 0,Y 370.318,Z 967.347,A -85,B 0,C 180,E1 -8029.232,E2 -8029.232} C_VEL
LIN {X 0,Y 371.884,Z 955.973,A -85,B 0,C 180,E1 -8032.35,E2 -8032.35} C_VEL
LIN {X 0,Y 373.984,Z 942.808,A -85,B 0,C 180,E1 -8035.358,E2 -8035.358} C_VEL
LIN {X 0,Y 376.733,Z 927.042,A -85,B 0,C 180,E1 -8038.364,E2 -8038.364} C_VEL
LIN {X 0,Y 379.872,Z 909.894,A -85,B 0,C 180,E1 -8041.106,E2 -8041.106} C_VEL
LIN {X 0,Y 383.185,Z 892.164,A -85,B 0,C 180,E1 -8043.495,E2 -8043.495} C_VEL
LIN {X 0,Y 386.947,Z 871.448,A -85,B 0,C 180,E1 -8045.822,E2 -8045.822} C_VEL
LIN {X 0,Y 390.381,Z 852.121,A -85,B 0,C 180,E1 -8047.651,E2 -8047.651} C_VEL
LIN {X 0,Y 393.704,Z 831.867,A -85,B 0,C 180,E1 -8049.233,E2 -8049.233} C_VEL
LIN {X 0,Y 397.06,Z 809.616,A -85,B 0,C 180,E1 -8050.653,E2 -8050.653} C_VEL
LIN {X 0,Y 399.953,Z 787.932,A -85,B 0,C 180,E1 -8051.754,E2 -8051.754} C_VEL
LIN {X 0,Y 402.417,Z 765.933,A -85,B 0,C 180,E1 -8052.602,E2 -8052.602} C_VEL
LIN {X 0,Y 404.234,Z 743.283,A -85,B 0,C 180,E1 -8053.236,E2 -8053.236} C_VEL
LIN {X 0,Y 405.869,Z 717.26,A -85,B 0,C 180,E1 -8053.78,E2 -8053.78} C_VEL
LIN {X 0,Y 407.051,Z 708.217,A -85,B 0,C 180,E1 -8053.941,E2 -8053.941} C_VEL
LIN {X 0,Y 416.953,Z 681.618,A -85,B 0,C 180,E1 -8055.219,E2 -8055.219} C_VEL
LIN {X 0,Y 425.39,Z 662.391,A -85,B 0,C 180,E1 -8055.991,E2 -8055.991} C_VEL
LIN {X 0,Y 431.754,Z 649.111,A -85,B 0,C 180,E1 -8056.456,E2 -8056.456} C_VEL
LIN {X 0,Y 441.315,Z 628.961,A -85,B 0,C 180,E1 -8057.132,E2 -8057.132} C_VEL
LIN {X 0,Y 447.504,Z 617.13,A -85,B 0,C 180,E1 -8057.457,E2 -8057.457} C_VEL
LIN {X 0,Y 439.358,Z 604.679,A -85,B 0,C 180,E1 -8059.394,E2 -8059.394} C_VEL
LIN {X 0,Y 432.384,Z 589.591,A -85,B 0,C 180,E1 -8061.535,E2 -8061.535} C_VEL
LIN {X 0,Y 427.634,Z 573.902,A -85,B 0,C 180,E1 -8063.568,E2 -8063.568} C_VEL
LIN {X 0,Y 424.731,Z 556.674,A -85,B 0,C 180,E1 -8065.599,E2 -8065.599} C_VEL
LIN {X 0,Y 423.697,Z 536.981,A -85,B 0,C 180,E1 -8067.69,E2 -8067.69} C_VEL
LIN {X 0,Y 424.628,Z 517.238,A -85,B 0,C 180,E1 -8069.586,E2 -8069.586} C_VEL
LIN {X 0,Y 428.069,Z 491.309,A -85,B 0,C 180,E1 -8071.798,E2 -8071.798} C_VEL
LIN {X 0,Y 428.395,Z 488.768,A -85,B 0,C 180,E1 -8072.023,E2 -8072.023} C_VEL
LIN {X 0,Y 419.301,Z 471.577,A -85,B 0,C 180,E1 -8075.486,E2 -8075.486} C_VEL
LIN {X 0,Y 410.349,Z 454.987,A -85,B 0,C 180,E1 -8079.161,E2 -8079.161} C_VEL
LIN {X 0,Y 401.971,Z 440.243,A -85,B 0,C 180,E1 -8082.783,E2 -8082.783} C_VEL
LIN {X 0,Y 395.773,Z 429.462,A -85,B 0,C 180,E1 -8085.666,E2 -8085.666} C_VEL
LIN {X 0,Y 390.654,Z 420.592,A -85,B 0,C 180,E1 -8088.185,E2 -8088.185} C_VEL
LIN {X 0,Y 386.697,Z 414.078,A -85,B 0,C 180,E1 -8090.175,E2 -8090.175} C_VEL
LIN {X 0,Y 384.566,Z 410.285,A -85,B 0,C 180,E1 -8091.327,E2 -8091.327} C_VEL
LIN {X 0,Y 381.637,Z 405.298,A -85,B 0,C 180,E1 -8092.927,E2 -8092.927} C_VEL
LIN {X 0,Y 378.622,Z 400.239,A -85,B 0,C 180,E1 -8094.604,E2 -8094.604} C_VEL
LIN {X 0,Y 376.392,Z 396.569,A -85,B 0,C 180,E1 -8095.887,E2 -8095.887} C_VEL
LIN {X 0,Y 375.673,Z 395.158,A -85,B 0,C 180,E1 -8096.338,E2 -8096.338} C_VEL
LIN {X 0,Y 373.322,Z 391.555,A -85,B 0,C 180,E1 -8097.698,E2 -8097.698} C_VEL
LIN {X 0,Y 372.744,Z 389.987,A -85,B 0,C 180,E1 -8098.156,E2 -8098.156} C_VEL
LIN {X 0,Y 370.465,Z 387.136,A -85,B 0,C 180,E1 -8099.382,E2 -8099.382} C_VEL
LIN {X 0,Y 369.734,Z 384.682,A -85,B 0,C 180,E1 -8100.155,E2 -8100.155} C_VEL
LIN {X 0,Y 369.726,Z 384.686,A -85,B 0,C 180,E1 -8104.499,E2 -8104.499} C_VEL
LIN {X 0,Y 369.722,Z 384.683,A -85,B 0,C 180,E1 -8108.398,E2 -8108.398} C_VEL
LIN {X 0,Y 369.734,Z 384.677,A -85,B 0,C 180,E1 -8112.653,E2 -8112.653} C_VEL
LIN {X 0,Y 369.716,Z 384.683,A -85,B 0,C 180,E1 -8116.497,E2 -8116.497} C_VEL
LIN {X 0,Y 369.739,Z 384.673,A -85,B 0,C 180,E1 -8120.748,E2 -8120.748} C_VEL
LIN {X 0,Y 369.708,Z 384.683,A -85,B 0,C 180,E1 -8124.784,E2 -8124.784} C_VEL
LIN {X 0,Y 369.746,Z 384.677,A -85,B 0,C 180,E1 -8128.951,E2 -8128.951} C_VEL
LIN {X 0,Y 369.706,Z 384.685,A -85,B 0,C 180,E1 -8133.031,E2 -8133.031} C_VEL
LIN {X 0,Y 369.737,Z 384.628,A -85,B 0,C 180,E1 -8137.089,E2 -8137.089} C_VEL
LIN {X 0,Y 369.728,Z 384.687,A -85,B 0,C 180,E1 -8140.172,E2 -8140.172} C_VEL
LIN {X 0,Y 370.978,Z 388.082,A -85,B 0,C 180,E1 -8140.711,E2 -8140.711} C_VEL
LIN {X 0,Y 372.4,Z 389.995,A -85,B 0,C 180,E1 -8141.133,E2 -8141.133} C_VEL
LIN {X 0,Y 379.68,Z 403.83,A -85,B 0,C 180,E1 -8143.627,E2 -8143.627} C_VEL
LIN {X 0,Y 387.548,Z 420.417,A -85,B 0,C 180,E1 -8146.36,E2 -8146.36} C_VEL
LIN {X 0,Y 394.605,Z 437.646,A -85,B 0,C 180,E1 -8148.922,E2 -8148.922} C_VEL
LIN {X 0,Y 398.527,Z 448.978,A -85,B 0,C 180,E1 -8150.46,E2 -8150.46} C_VEL
LIN {X 0,Y 396.347,Z 490.466,A -85,B 0,C 180,E1 -8153.732,E2 -8153.732} C_VEL
LIN {X 0,Y 396.16,Z 500.489,A -85,B 0,C 180,E1 -8154.438,E2 -8154.438} C_VEL
LIN {X 0,Y 396.98,Z 508.379,A -85,B 0,C 180,E1 -8154.7,E2 -8154.7} C_VEL
LIN {X 0,Y 391.383,Z 705.291,A -85,B 0,C 180,E1 -8158.435,E2 -8158.435} C_VEL
LIN {X 0,Y 390.783,Z 723.938,A -85,B 0,C 180,E1 -8159.017,E2 -8159.017} C_VEL
LIN {X 0,Y 389.705,Z 741.941,A -85,B 0,C 180,E1 -8159.842,E2 -8159.842} C_VEL
LIN {X 0,Y 388.101,Z 759.91,A -85,B 0,C 180,E1 -8160.947,E2 -8160.947} C_VEL
LIN {X 0,Y 386.135,Z 777.033,A -85,B 0,C 180,E1 -8162.303,E2 -8162.303} C_VEL
LIN {X 0,Y 383.96,Z 793.02,A -85,B 0,C 180,E1 -8163.891,E2 -8163.891} C_VEL
LIN {X 0,Y 381.697,Z 807.348,A -85,B 0,C 180,E1 -8165.634,E2 -8165.634} C_VEL
LIN {X 0,Y 379.462,Z 820.283,A -85,B 0,C 180,E1 -8167.539,E2 -8167.539} C_VEL
LIN {X 0,Y 377.258,Z 832.348,A -85,B 0,C 180,E1 -8169.685,E2 -8169.685} C_VEL
LIN {X 0,Y 375.176,Z 843.358,A -85,B 0,C 180,E1 -8172.069,E2 -8172.069} C_VEL
LIN {X 0,Y 373.393,Z 852.924,A -85,B 0,C 180,E1 -8174.628,E2 -8174.628} C_VEL
LIN {X 0,Y 373.131,Z 854.34,A -85,B 0,C 180,E1 -8175.064,E2 -8175.064} C_VEL
LIN {X 0,Y 371.566,Z 857.84,A -85,B 0,C 180,E1 -8176.11,E2 -8176.11} C_VEL
LIN {X 0,Y 364.479,Z 866.021,A -85,B 0,C 180,E1 -8178.75,E2 -8178.75} C_VEL
LIN {X 0,Y 363.087,Z 868.537,A -85,B 0,C 180,E1 -8179.887,E2 -8179.887} C_VEL
LIN {X 0,Y 362.324,Z 873.337,A -85,B 0,C 180,E1 -8182.867,E2 -8182.867} C_VEL
LIN {X 0,Y 361.889,Z 876.43,A -85,B 0,C 180,E1 -8185.881,E2 -8185.881} C_VEL
LIN {X 0,Y 361.698,Z 877.863,A -85,B 0,C 180,E1 -8188.892,E2 -8188.892} C_VEL
LIN {X 0,Y 361.727,Z 877.671,A -85,B 0,C 180,E1 -8191.901,E2 -8191.901} C_VEL
LIN {X 0,Y 361.97,Z 875.85,A -85,B 0,C 180,E1 -8194.913,E2 -8194.913} C_VEL
LIN {X 0,Y 362.467,Z 872.341,A -85,B 0,C 180,E1 -8197.928,E2 -8197.928} C_VEL
LIN {X 0,Y 363.338,Z 867.025,A -85,B 0,C 180,E1 -8200.946,E2 -8200.946} C_VEL
LIN {X 0,Y 364.609,Z 860.16,A -85,B 0,C 180,E1 -8203.803,E2 -8203.803} C_VEL
LIN {X 0,Y 366.226,Z 851.827,A -85,B 0,C 180,E1 -8206.496,E2 -8206.496} C_VEL
LIN {X 0,Y 368.172,Z 842.065,A -85,B 0,C 180,E1 -8209.02,E2 -8209.02} C_VEL
LIN {X 0,Y 370.402,Z 830.891,A -85,B 0,C 180,E1 -8211.372,E2 -8211.372} C_VEL
LIN {X 0,Y 372.802,Z 818.27,A -85,B 0,C 180,E1 -8213.555,E2 -8213.555} C_VEL
LIN {X 0,Y 375.327,Z 804.082,A -85,B 0,C 180,E1 -8215.567,E2 -8215.567} C_VEL
LIN {X 0,Y 377.718,Z 789.081,A -85,B 0,C 180,E1 -8217.305,E2 -8217.305} C_VEL
LIN {X 0,Y 379.848,Z 773.266,A -85,B 0,C 180,E1 -8218.797,E2 -8218.797} C_VEL
LIN {X 0,Y 381.822,Z 755.826,A -85,B 0,C 180,E1 -8220.098,E2 -8220.098} C_VEL
LIN {X 0,Y 383.317,Z 737.832,A -85,B 0,C 180,E1 -8221.131,E2 -8221.131} C_VEL
LIN {X 0,Y 384.309,Z 719.504,A -85,B 0,C 180,E1 -8221.897,E2 -8221.897} C_VEL
LIN {X 0,Y 384.79,Z 699.798,A -85,B 0,C 180,E1 -8222.437,E2 -8222.437} C_VEL
LIN {X 0,Y 390.466,Z 507.074,A -85,B 0,C 180,E1 -8226.14,E2 -8226.14} C_VEL
LIN {X 0,Y 389.688,Z 499.945,A -85,B 0,C 180,E1 -8226.441,E2 -8226.441} C_VEL
LIN {X 0,Y 391.537,Z 461.925,A -85,B 0,C 180,E1 -8229.39,E2 -8229.39} C_VEL
LIN {X 0,Y 392.129,Z 451.963,A -85,B 0,C 180,E1 -8230.21,E2 -8230.21} C_VEL
LIN {X 0,Y 385.263,Z 433.65,A -85,B 0,C 180,E1 -8232.841,E2 -8232.841} C_VEL
LIN {X 0,Y 384.126,Z 431.435,A -85,B 0,C 180,E1 -8233.211,E2 -8233.211} C_VEL
LIN {X 0,Y 383.284,Z 431.138,A -85,B 0,C 180,E1 -8233.398,E2 -8233.398} C_VEL
LIN {X 0,Y 390.124,Z 448.123,A -85,B 0,C 180,E1 -8236.495,E2 -8236.495} C_VEL
LIN {X 0,Y 394.174,Z 459.158,A -85,B 0,C 180,E1 -8238.349,E2 -8238.349} C_VEL
LIN {X 0,Y 389.172,Z 499.934,A -85,B 0,C 180,E1 -8242.397,E2 -8242.397} C_VEL
LIN {X 0,Y 384.29,Z 543.314,A -85,B 0,C 180,E1 -8246.636,E2 -8246.636} C_VEL
LIN {X 0,Y 379.734,Z 588.642,A -85,B 0,C 180,E1 -8251.021,E2 -8251.021} C_VEL
LIN {X 0,Y 378.082,Z 607.88,A -85,B 0,C 180,E1 -8252.831,E2 -8252.831} C_VEL
LIN {X 0,Y 378.723,Z 617.613,A -85,B 0,C 180,E1 -8253.189,E2 -8253.189} C_VEL
LIN {X 0,Y 372.235,Z 752.117,A -85,B 0,C 180,E1 -8256.927,E2 -8256.927} C_VEL
LIN {X 0,Y 371.602,Z 769.119,A -85,B 0,C 180,E1 -8257.621,E2 -8257.621} C_VEL
LIN {X 0,Y 370.591,Z 786.294,A -85,B 0,C 180,E1 -8258.639,E2 -8258.639} C_VEL
LIN {X 0,Y 369.475,Z 801.282,A -85,B 0,C 180,E1 -8259.816,E2 -8259.816} C_VEL
LIN {X 0,Y 368.081,Z 816.866,A -85,B 0,C 180,E1 -8261.386,E2 -8261.386} C_VEL
LIN {X 0,Y 366.791,Z 829.946,A -85,B 0,C 180,E1 -8263.041,E2 -8263.041} C_VEL
LIN {X 0,Y 365.528,Z 842.104,A -85,B 0,C 180,E1 -8264.938,E2 -8264.938} C_VEL
LIN {X 0,Y 364.423,Z 852.783,A -85,B 0,C 180,E1 -8266.998,E2 -8266.998} C_VEL
LIN {X 0,Y 363.46,Z 862.643,A -85,B 0,C 180,E1 -8269.378,E2 -8269.378} C_VEL
LIN {X 0,Y 362.792,Z 870.278,A -85,B 0,C 180,E1 -8271.76,E2 -8271.76} C_VEL
LIN {X 0,Y 362.377,Z 876.438,A -85,B 0,C 180,E1 -8274.299,E2 -8274.299} C_VEL
LIN {X 0,Y 362.221,Z 880.862,A -85,B 0,C 180,E1 -8276.993,E2 -8276.993} C_VEL
LIN {X 0,Y 362.295,Z 883.313,A -85,B 0,C 180,E1 -8279.525,E2 -8279.525} C_VEL
LIN {X 0,Y 362.59,Z 884.043,A -85,B 0,C 180,E1 -8282.212,E2 -8282.212} C_VEL
LIN {X 0,Y 363.115,Z 883.041,A -85,B 0,C 180,E1 -8284.738,E2 -8284.738} C_VEL
LIN {X 0,Y 363.982,Z 880.157,A -85,B 0,C 180,E1 -8287.418,E2 -8287.418} C_VEL
LIN {X 0,Y 365.15,Z 875.571,A -85,B 0,C 180,E1 -8289.933,E2 -8289.933} C_VEL
LIN {X 0,Y 366.617,Z 869.594,A -85,B 0,C 180,E1 -8292.282,E2 -8292.282} C_VEL
LIN {X 0,Y 368.401,Z 861.602,A -85,B 0,C 180,E1 -8294.62,E2 -8294.62} C_VEL
LIN {X 0,Y 370.297,Z 852.903,A -85,B 0,C 180,E1 -8296.631,E2 -8296.631} C_VEL
LIN {X 0,Y 372.66,Z 841.107,A -85,B 0,C 180,E1 -8298.781,E2 -8298.781} C_VEL
LIN {X 0,Y 375.046,Z 827.913,A -85,B 0,C 180,E1 -8300.677,E2 -8300.677} C_VEL
LIN {X 0,Y 377.386,Z 813.11,A -85,B 0,C 180,E1 -8302.353,E2 -8302.353} C_VEL
LIN {X 0,Y 379.514,Z 797.015,A -85,B 0,C 180,E1 -8303.771,E2 -8303.771} C_VEL
LIN {X 0,Y 381.452,Z 779.232,A -85,B 0,C 180,E1 -8304.961,E2 -8304.961} C_VEL
LIN {X 0,Y 385.458,Z 752.558,A -85,B 0,C 180,E1 -8306.497,E2 -8306.497} C_VEL
LIN {X 0,Y 396.212,Z 701.288,A -85,B 0,C 180,E1 -8309.063,E2 -8309.063} C_VEL
LIN {X 0,Y 406.045,Z 652.955,A -85,B 0,C 180,E1 -8311.097,E2 -8311.097} C_VEL
LIN {X 0,Y 413.575,Z 638.092,A -85,B 0,C 180,E1 -8312.05,E2 -8312.05} C_VEL
LIN {X 0,Y 423.449,Z 617.812,A -85,B 0,C 180,E1 -8314.684,E2 -8314.684} C_VEL
LIN {X 0,Y 434.203,Z 601.326,A -85,B 0,C 180,E1 -8316.942,E2 -8316.942} C_VEL
LIN {X 0,Y 435.976,Z 599.035,A -85,B 0,C 180,E1 -8317.268,E2 -8317.268} C_VEL
LIN {X 0,Y 435.051,Z 605.902,A -85,B 0,C 180,E1 -8319.03,E2 -8319.03} C_VEL
LIN {X 0,Y 436.312,Z 613.29,A -85,B 0,C 180,E1 -8320.866,E2 -8320.866} C_VEL
LIN {X 0,Y 438.734,Z 619.094,A -85,B 0,C 180,E1 -8322.236,E2 -8322.236} C_VEL
LIN {X 0,Y 428.262,Z 640.096,A -85,B 0,C 180,E1 -8322.853,E2 -8322.853} C_VEL
LIN {X 0,Y 421.607,Z 654.482,A -85,B 0,C 180,E1 -8323.374,E2 -8323.374} C_VEL
LIN {X 0,Y 412.654,Z 673.96,A -85,B 0,C 180,E1 -8324.075,E2 -8324.075} C_VEL
LIN {X 0,Y 405.878,Z 691.275,A -85,B 0,C 180,E1 -8324.851,E2 -8324.851} C_VEL
LIN {X 0,Y 400.51,Z 725.804,A -85,B 0,C 180,E1 -8325.52,E2 -8325.52} C_VEL
LIN {X 0,Y 397.017,Z 752.846,A -85,B 0,C 180,E1 -8326.439,E2 -8326.439} C_VEL
LIN {X 0,Y 392.911,Z 779.299,A -85,B 0,C 180,E1 -8327.595,E2 -8327.595} C_VEL
LIN {X 0,Y 388.633,Z 804.936,A -85,B 0,C 180,E1 -8329.056,E2 -8329.056} C_VEL
LIN {X 0,Y 384.578,Z 828.611,A -85,B 0,C 180,E1 -8330.722,E2 -8330.722} C_VEL
LIN {X 0,Y 380.468,Z 851.903,A -85,B 0,C 180,E1 -8332.717,E2 -8332.717} C_VEL
LIN {X 0,Y 376.637,Z 873.861,A -85,B 0,C 180,E1 -8334.957,E2 -8334.957} C_VEL
LIN {X 0,Y 373.088,Z 894.137,A -85,B 0,C 180,E1 -8337.406,E2 -8337.406} C_VEL
LIN {X 0,Y 369.808,Z 913.442,A -85,B 0,C 180,E1 -8340.166,E2 -8340.166} C_VEL
LIN {X 0,Y 367.134,Z 929.91,A -85,B 0,C 180,E1 -8342.947,E2 -8342.947} C_VEL
LIN {X 0,Y 364.898,Z 944.719,A -85,B 0,C 180,E1 -8345.903,E2 -8345.903} C_VEL
LIN {X 0,Y 363.213,Z 957.237,A -85,B 0,C 180,E1 -8348.861,E2 -8348.861} C_VEL
LIN {X 0,Y 361.949,Z 968.255,A -85,B 0,C 180,E1 -8351.977,E2 -8351.977} C_VEL
LIN {X 0,Y 361.099,Z 977.657,A -85,B 0,C 180,E1 -8355.241,E2 -8355.241} C_VEL
LIN {X 0,Y 360.683,Z 985.003,A -85,B 0,C 180,E1 -8358.486,E2 -8358.486} C_VEL
LIN {X 0,Y 360.517,Z 990.269,A -85,B 0,C 180,E1 -8361.547,E2 -8361.547} C_VEL
LIN {X 0,Y 360.497,Z 994.06,A -85,B 0,C 180,E1 -8364.748,E2 -8364.748} C_VEL
LIN {X 0,Y 360.517,Z 996.088,A -85,B 0,C 180,E1 -8367.774,E2 -8367.774} C_VEL
LIN {X 0,Y 360.506,Z 996.602,A -85,B 0,C 180,E1 -8370.953,E2 -8370.953} C_VEL
LIN {X 0,Y 360.455,Z 995.553,A -85,B 0,C 180,E1 -8373.976,E2 -8373.976} C_VEL
LIN {X 0,Y 360.384,Z 992.841,A -85,B 0,C 180,E1 -8377.172,E2 -8377.172} C_VEL
LIN {X 0,Y 360.458,Z 988.697,A -85,B 0,C 180,E1 -8380.225,E2 -8380.225} C_VEL
LIN {X 0,Y 360.767,Z 982.666,A -85,B 0,C 180,E1 -8383.462,E2 -8383.462} C_VEL
LIN {X 0,Y 361.502,Z 974.322,A -85,B 0,C 180,E1 -8386.882,E2 -8386.882} C_VEL
LIN {X 0,Y 362.705,Z 964.316,A -85,B 0,C 180,E1 -8390.156,E2 -8390.156} C_VEL
LIN {X 0,Y 364.418,Z 952.739,A -85,B 0,C 180,E1 -8393.271,E2 -8393.271} C_VEL
LIN {X 0,Y 366.633,Z 939.681,A -85,B 0,C 180,E1 -8396.218,E2 -8396.218} C_VEL
LIN {X 0,Y 369.343,Z 924.946,A -85,B 0,C 180,E1 -8399.027,E2 -8399.027} C_VEL
LIN {X 0,Y 372.503,Z 908.385,A -85,B 0,C 180,E1 -8401.693,E2 -8401.693} C_VEL
LIN {X 0,Y 375.985,Z 890.459,A -85,B 0,C 180,E1 -8404.132,E2 -8404.132} C_VEL
LIN {X 0,Y 379.794,Z 870.336,A -85,B 0,C 180,E1 -8406.417,E2 -8406.417} C_VEL
LIN {X 0,Y 383.385,Z 850.846,A -85,B 0,C 180,E1 -8408.28,E2 -8408.28} C_VEL
LIN {X 0,Y 386.806,Z 830.685,A -85,B 0,C 180,E1 -8409.87,E2 -8409.87} C_VEL
LIN {X 0,Y 390.155,Z 809.396,A -85,B 0,C 180,E1 -8411.251,E2 -8411.251} C_VEL
LIN {X 0,Y 393.163,Z 787.884,A -85,B 0,C 180,E1 -8412.37,E2 -8412.37} C_VEL
LIN {X 0,Y 395.79,Z 765.394,A -85,B 0,C 180,E1 -8413.254,E2 -8413.254} C_VEL
LIN {X 0,Y 397.715,Z 742.48,A -85,B 0,C 180,E1 -8413.91,E2 -8413.91} C_VEL
LIN {X 0,Y 399.392,Z 717.097,A -85,B 0,C 180,E1 -8414.448,E2 -8414.448} C_VEL
LIN {X 0,Y 400.687,Z 707.503,A -85,B 0,C 180,E1 -8414.623,E2 -8414.623} C_VEL
LIN {X 0,Y 411.088,Z 680,A -85,B 0,C 180,E1 -8415.949,E2 -8415.949} C_VEL
LIN {X 0,Y 419.813,Z 660.435,A -85,B 0,C 180,E1 -8416.726,E2 -8416.726} C_VEL
LIN {X 0,Y 426.098,Z 647.37,A -85,B 0,C 180,E1 -8417.181,E2 -8417.181} C_VEL
LIN {X 0,Y 436.109,Z 626.696,A -85,B 0,C 180,E1 -8417.874,E2 -8417.874} C_VEL
LIN {X 0,Y 439.684,Z 619.711,A -85,B 0,C 180,E1 -8418.083,E2 -8418.083} C_VEL
LIN {X 0,Y 432.2,Z 607.429,A -85,B 0,C 180,E1 -8419.975,E2 -8419.975} C_VEL
LIN {X 0,Y 425.462,Z 591.904,A -85,B 0,C 180,E1 -8422.167,E2 -8422.167} C_VEL
LIN {X 0,Y 420.964,Z 575.777,A -85,B 0,C 180,E1 -8424.248,E2 -8424.248} C_VEL
LIN {X 0,Y 418.324,Z 558.122,A -85,B 0,C 180,E1 -8426.323,E2 -8426.323} C_VEL
LIN {X 0,Y 417.637,Z 538.086,A -85,B 0,C 180,E1 -8428.462,E2 -8428.462} C_VEL
LIN {X 0,Y 418.844,Z 517.98,A -85,B 0,C 180,E1 -8430.387,E2 -8430.387} C_VEL
LIN {X 0,Y 422.321,Z 493.017,A -85,B 0,C 180,E1 -8432.544,E2 -8432.544} C_VEL
LIN {X 0,Y 414.006,Z 477.238,A -85,B 0,C 180,E1 -8435.76,E2 -8435.76} C_VEL
LIN {X 0,Y 405.043,Z 460.566,A -85,B 0,C 180,E1 -8439.481,E2 -8439.481} C_VEL
LIN {X 0,Y 396.999,Z 446.303,A -85,B 0,C 180,E1 -8443.014,E2 -8443.014} C_VEL
LIN {X 0,Y 390.507,Z 434.967,A -85,B 0,C 180,E1 -8446.074,E2 -8446.074} C_VEL
LIN {X 0,Y 385.05,Z 425.642,A -85,B 0,C 180,E1 -8448.77,E2 -8448.77} C_VEL
LIN {X 0,Y 379.814,Z 416.589,A -85,B 0,C 180,E1 -8451.523,E2 -8451.523} C_VEL
LIN {X 0,Y 376.489,Z 411.067,A -85,B 0,C 180,E1 -8453.336,E2 -8453.336} C_VEL
LIN {X 0,Y 373.7,Z 406.304,A -85,B 0,C 180,E1 -8454.935,E2 -8454.935} C_VEL
LIN {X 0,Y 370.535,Z 401.041,A -85,B 0,C 180,E1 -8456.769,E2 -8456.769} C_VEL
LIN {X 0,Y 368.332,Z 397.186,A -85,B 0,C 180,E1 -8458.134,E2 -8458.134} C_VEL
LIN {X 0,Y 367.244,Z 395.607,A -85,B 0,C 180,E1 -8458.752,E2 -8458.752} C_VEL
LIN {X 0,Y 365.315,Z 392.28,A -85,B 0,C 180,E1 -8460,E2 -8460} C_VEL
LIN {X 0,Y 364.653,Z 390.863,A -85,B 0,C 180,E1 -8460.472,E2 -8460.472} C_VEL
LIN {X 0,Y 362.257,Z 387.595,A -85,B 0,C 180,E1 -8461.898,E2 -8461.898} C_VEL
LIN {X 0,Y 361.767,Z 385.675,A -85,B 0,C 180,E1 -8462.456,E2 -8462.456} C_VEL
LIN {X 0,Y 361.807,Z 385.676,A -85,B 0,C 180,E1 -8466.506,E2 -8466.506} C_VEL
LIN {X 0,Y 361.771,Z 385.67,A -85,B 0,C 180,E1 -8470.672,E2 -8470.672} C_VEL
LIN {X 0,Y 361.801,Z 385.666,A -85,B 0,C 180,E1 -8474.729,E2 -8474.729} C_VEL
LIN {X 0,Y 361.784,Z 385.668,A -85,B 0,C 180,E1 -8479.06,E2 -8479.06} C_VEL
LIN {X 0,Y 361.79,Z 385.667,A -85,B 0,C 180,E1 -8483.107,E2 -8483.107} C_VEL
LIN {X 0,Y 361.803,Z 385.652,A -85,B 0,C 180,E1 -8487.49,E2 -8487.49} C_VEL
LIN {X 0,Y 361.781,Z 385.656,A -85,B 0,C 180,E1 -8491.49,E2 -8491.49} C_VEL
LIN {X 0,Y 361.798,Z 385.619,A -85,B 0,C 180,E1 -8495.671,E2 -8495.671} C_VEL
LIN {X 0,Y 361.807,Z 385.759,A -85,B 0,C 180,E1 -8498.853,E2 -8498.853} C_VEL
LIN {X 0,Y 362.817,Z 388.741,A -85,B 0,C 180,E1 -8499.335,E2 -8499.335} C_VEL
LIN {X 0,Y 364.649,Z 391.262,A -85,B 0,C 180,E1 -8499.913,E2 -8499.913} C_VEL
LIN {X 0,Y 366.765,Z 395.097,A -85,B 0,C 180,E1 -8500.659,E2 -8500.659} C_VEL
LIN {X 0,Y 374.376,Z 409.573,A -85,B 0,C 180,E1 -8503.345,E2 -8503.345} C_VEL
LIN {X 0,Y 381.947,Z 425.771,A -85,B 0,C 180,E1 -8506.046,E2 -8506.046} C_VEL
LIN {X 0,Y 388.909,Z 443.04,A -85,B 0,C 180,E1 -8508.653,E2 -8508.653} C_VEL
LIN {X 0,Y 392.101,Z 452.063,A -85,B 0,C 180,E1 -8509.908,E2 -8509.908} C_VEL
LIN {X 0,Y 389.769,Z 495.822,A -85,B 0,C 180,E1 -8513.357,E2 -8513.357} C_VEL
LIN {X 0,Y 389.739,Z 501.868,A -85,B 0,C 180,E1 -8513.765,E2 -8513.765} C_VEL
LIN {X 0,Y 390.515,Z 509.589,A -85,B 0,C 180,E1 -8514.027,E2 -8514.027} C_VEL
LIN {X 0,Y 384.654,Z 706.082,A -85,B 0,C 180,E1 -8517.806,E2 -8517.806} C_VEL
LIN {X 0,Y 384.045,Z 724.593,A -85,B 0,C 180,E1 -8518.387,E2 -8518.387} C_VEL
LIN {X 0,Y 382.929,Z 742.653,A -85,B 0,C 180,E1 -8519.219,E2 -8519.219} C_VEL
LIN {X 0,Y 381.33,Z 760.076,A -85,B 0,C 180,E1 -8520.294,E2 -8520.294} C_VEL
LIN {X 0,Y 379.266,Z 777.423,A -85,B 0,C 180,E1 -8521.671,E2 -8521.671} C_VEL
LIN {X 0,Y 376.984,Z 793.574,A -85,B 0,C 180,E1 -8523.285,E2 -8523.285} C_VEL
LIN {X 0,Y 374.607,Z 808.027,A -85,B 0,C 180,E1 -8525.058,E2 -8525.058} C_VEL
LIN {X 0,Y 372.161,Z 821.544,A -85,B 0,C 180,E1 -8527.073,E2 -8527.073} C_VEL
LIN {X 0,Y 369.786,Z 833.91,A -85,B 0,C 180,E1 -8529.317,E2 -8529.317} C_VEL
LIN {X 0,Y 367.58,Z 844.971,A -85,B 0,C 180,E1 -8531.772,E2 -8531.772} C_VEL
LIN {X 0,Y 365.661,Z 854.724,A -85,B 0,C 180,E1 -8534.457,E2 -8534.457} C_VEL
LIN {X 0,Y 364.099,Z 862.841,A -85,B 0,C 180,E1 -8537.31,E2 -8537.31} C_VEL
LIN {X 0,Y 363.087,Z 868.537,A -85,B 0,C 180,E1 -8539.887,E2 -8539.887} C_VEL
LIN {X 0,Y 361.751,Z 870.817,A -85,B 0,C 180,E1 -8541.045,E2 -8541.045} C_VEL
LIN {X 0,Y 355.08,Z 876.042,A -85,B 0,C 180,E1 -8544.068,E2 -8544.068} C_VEL
LIN {X 0,Y 354.076,Z 877.229,A -85,B 0,C 180,E1 -8545.207,E2 -8545.207} C_VEL
LIN {X 0,Y 353.821,Z 879.022,A -85,B 0,C 180,E1 -8548.381,E2 -8548.381} C_VEL
LIN {X 0,Y 353.81,Z 879.099,A -85,B 0,C 180,E1 -8551.458,E2 -8551.458} C_VEL
LIN {X 0,Y 354.04,Z 877.548,A -85,B 0,C 180,E1 -8554.536,E2 -8554.536} C_VEL
LIN {X 0,Y 354.525,Z 874.313,A -85,B 0,C 180,E1 -8557.618,E2 -8557.618} C_VEL
LIN {X 0,Y 355.389,Z 869.275,A -85,B 0,C 180,E1 -8560.702,E2 -8560.702} C_VEL
LIN {X 0,Y 356.659,Z 862.711,A -85,B 0,C 180,E1 -8563.621,E2 -8563.621} C_VEL
LIN {X 0,Y 358.294,Z 854.706,A -85,B 0,C 180,E1 -8566.371,E2 -8566.371} C_VEL
LIN {X 0,Y 360.269,Z 845.31,A -85,B 0,C 180,E1 -8568.949,E2 -8568.949} C_VEL
LIN {X 0,Y 362.539,Z 834.551,A -85,B 0,C 180,E1 -8571.349,E2 -8571.349} C_VEL
LIN {X 0,Y 364.989,Z 822.414,A -85,B 0,C 180,E1 -8573.576,E2 -8573.576} C_VEL
LIN {X 0,Y 367.672,Z 808.23,A -85,B 0,C 180,E1 -8575.706,E2 -8575.706} C_VEL
LIN {X 0,Y 370.294,Z 792.842,A -85,B 0,C 180,E1 -8577.587,E2 -8577.587} C_VEL
LIN {X 0,Y 372.582,Z 777.097,A -85,B 0,C 180,E1 -8579.149,E2 -8579.149} C_VEL
LIN {X 0,Y 374.631,Z 760.415,A -85,B 0,C 180,E1 -8580.471,E2 -8580.471} C_VEL
LIN {X 0,Y 376.296,Z 742.688,A -85,B 0,C 180,E1 -8581.565,E2 -8581.565} C_VEL
LIN {X 0,Y 377.46,Z 724.111,A -85,B 0,C 180,E1 -8582.412,E2 -8582.412} C_VEL
LIN {X 0,Y 378.062,Z 704.971,A -85,B 0,C 180,E1 -8582.992,E2 -8582.992} C_VEL
LIN {X 0,Y 384.057,Z 508.208,A -85,B 0,C 180,E1 -8586.84,E2 -8586.84} C_VEL
LIN {X 0,Y 383.293,Z 501.73,A -85,B 0,C 180,E1 -8587.103,E2 -8587.103} C_VEL
LIN {X 0,Y 385.235,Z 463.747,A -85,B 0,C 180,E1 -8590.067,E2 -8590.067} C_VEL
LIN {X 0,Y 385.622,Z 455.179,A -85,B 0,C 180,E1 -8590.789,E2 -8590.789} C_VEL
LIN {X 0,Y 379.441,Z 438.537,A -85,B 0,C 180,E1 -8593.23,E2 -8593.23} C_VEL
LIN {X 0,Y 378.153,Z 438.129,A -85,B 0,C 180,E1 -8593.508,E2 -8593.508} C_VEL
LIN {X 0,Y 384.733,Z 454.963,A -85,B 0,C 180,E1 -8596.584,E2 -8596.584} C_VEL
LIN {X 0,Y 387.535,Z 462.616,A -85,B 0,C 180,E1 -8597.87,E2 -8597.87} C_VEL
LIN {X 0,Y 382.292,Z 503.494,A -85,B 0,C 180,E1 -8601.97,E2 -8601.97} C_VEL
LIN {X 0,Y 377.193,Z 546.885,A -85,B 0,C 180,E1 -8606.265,E2 -8606.265} C_VEL
LIN {X 0,Y 372.405,Z 592.834,A -85,B 0,C 180,E1 -8610.761,E2 -8610.761} C_VEL
LIN {X 0,Y 371.002,Z 608.852,A -85,B 0,C 180,E1 -8612.274,E2 -8612.274} C_VEL
LIN {X 0,Y 371.612,Z 618.555,A -85,B 0,C 180,E1 -8612.639,E2 -8612.639} C_VEL
LIN {X 0,Y 364.775,Z 752.308,A -85,B 0,C 180,E1 -8616.478,E2 -8616.478} C_VEL
LIN {X 0,Y 364.081,Z 770.132,A -85,B 0,C 180,E1 -8617.218,E2 -8617.218} C_VEL
LIN {X 0,Y 363.029,Z 787.279,A -85,B 0,C 180,E1 -8618.257,E2 -8618.257} C_VEL
LIN {X 0,Y 361.87,Z 802.289,A -85,B 0,C 180,E1 -8619.457,E2 -8619.457} C_VEL
LIN {X 0,Y 360.421,Z 817.89,A -85,B 0,C 180,E1 -8621.06,E2 -8621.06} C_VEL
LIN {X 0,Y 359.062,Z 831.184,A -85,B 0,C 180,E1 -8622.774,E2 -8622.774} C_VEL
LIN {X 0,Y 357.718,Z 843.683,A -85,B 0,C 180,E1 -8624.767,E2 -8624.767} C_VEL
LIN {X 0,Y 356.574,Z 854.3,A -85,B 0,C 180,E1 -8626.871,E2 -8626.871} C_VEL
LIN {X 0,Y 355.58,Z 864.127,A -85,B 0,C 180,E1 -8629.304,E2 -8629.304} C_VEL
LIN {X 0,Y 354.894,Z 871.733,A -85,B 0,C 180,E1 -8631.738,E2 -8631.738} C_VEL
LIN {X 0,Y 354.474,Z 877.891,A -85,B 0,C 180,E1 -8634.334,E2 -8634.334} C_VEL
LIN {X 0,Y 354.328,Z 882.335,A -85,B 0,C 180,E1 -8637.088,E2 -8637.088} C_VEL
LIN {X 0,Y 354.428,Z 884.776,A -85,B 0,C 180,E1 -8639.676,E2 -8639.676} C_VEL
LIN {X 0,Y 354.762,Z 885.533,A -85,B 0,C 180,E1 -8642.422,E2 -8642.422} C_VEL
LIN {X 0,Y 355.35,Z 884.536,A -85,B 0,C 180,E1 -8645.004,E2 -8645.004} C_VEL
LIN {X 0,Y 356.306,Z 881.684,A -85,B 0,C 180,E1 -8647.741,E2 -8647.741} C_VEL
LIN {X 0,Y 357.594,Z 877.138,A -85,B 0,C 180,E1 -8650.308,E2 -8650.308} C_VEL
LIN {X 0,Y 359.179,Z 871.183,A -85,B 0,C 180,E1 -8652.704,E2 -8652.704} C_VEL
LIN {X 0,Y 361.274,Z 862.723,A -85,B 0,C 180,E1 -8655.243,E2 -8655.243} C_VEL
LIN {X 0,Y 363.679,Z 852.393,A -85,B 0,C 180,E1 -8657.603,E2 -8657.603} C_VEL
LIN {X 0,Y 365.916,Z 841.983,A -85,B 0,C 180,E1 -8659.487,E2 -8659.487} C_VEL
LIN {X 0,Y 368.393,Z 829.455,A -85,B 0,C 180,E1 -8661.327,E2 -8661.327} C_VEL
LIN {X 0,Y 370.904,Z 815.026,A -85,B 0,C 180,E1 -8663.009,E2 -8663.009} C_VEL
LIN {X 0,Y 373.244,Z 799.34,A -85,B 0,C 180,E1 -8664.448,E2 -8664.448} C_VEL
LIN {X 0,Y 375.55,Z 781.389,A -85,B 0,C 180,E1 -8665.719,E2 -8665.719} C_VEL
LIN {X 0,Y 380.356,Z 754.169,A -85,B 0,C 180,E1 -8667.389,E2 -8667.389} C_VEL
LIN {X 0,Y 390.851,Z 709.111,A -85,B 0,C 180,E1 -8669.754,E2 -8669.754} C_VEL
LIN {X 0,Y 399.652,Z 669.4,A -85,B 0,C 180,E1 -8671.515,E2 -8671.515} C_VEL
LIN {X 0,Y 402.78,Z 655.283,A -85,B 0,C 180,E1 -8672.088,E2 -8672.088} C_VEL
LIN {X 0,Y 410.403,Z 641.148,A -85,B 0,C 180,E1 -8672.991,E2 -8672.991} C_VEL
LIN {X 0,Y 420.482,Z 622.552,A -85,B 0,C 180,E1 -8675.464,E2 -8675.464} C_VEL
LIN {X 0,Y 431.057,Z 607.715,A -85,B 0,C 180,E1 -8677.55,E2 -8677.55} C_VEL
LIN {X 0,Y 430.682,Z 615.393,A -85,B 0,C 180,E1 -8679.577,E2 -8679.577} C_VEL
LIN {X 0,Y 432.684,Z 622.667,A -85,B 0,C 180,E1 -8681.421,E2 -8681.421} C_VEL
LIN {X 0,Y 422.224,Z 643.63,A -85,B 0,C 180,E1 -8682.079,E2 -8682.079} C_VEL
LIN {X 0,Y 416.405,Z 655.903,A -85,B 0,C 180,E1 -8682.509,E2 -8682.509} C_VEL
LIN {X 0,Y 407.051,Z 676.057,A -85,B 0,C 180,E1 -8683.26,E2 -8683.26} C_VEL
LIN {X 0,Y 402.03,Z 688.771,A -85,B 0,C 180,E1 -8683.843,E2 -8683.843} C_VEL
LIN {X 0,Y 395.761,Z 726.051,A -85,B 0,C 180,E1 -8684.593,E2 -8684.593} C_VEL
LIN {X 0,Y 391.228,Z 756.14,A -85,B 0,C 180,E1 -8685.69,E2 -8685.69} C_VEL
LIN {X 0,Y 386.573,Z 782.395,A -85,B 0,C 180,E1 -8686.934,E2 -8686.934} C_VEL
LIN {X 0,Y 382.241,Z 806.128,A -85,B 0,C 180,E1 -8688.362,E2 -8688.362} C_VEL
LIN {X 0,Y 377.669,Z 830.277,A -85,B 0,C 180,E1 -8690.157,E2 -8690.157} C_VEL
LIN {X 0,Y 373.219,Z 853.713,A -85,B 0,C 180,E1 -8692.254,E2 -8692.254} C_VEL
LIN {X 0,Y 369.14,Z 875.345,A -85,B 0,C 180,E1 -8694.574,E2 -8694.574} C_VEL
LIN {X 0,Y 365.511,Z 894.735,A -85,B 0,C 180,E1 -8697.018,E2 -8697.018} C_VEL
LIN {X 0,Y 362.281,Z 912.663,A -85,B 0,C 180,E1 -8699.664,E2 -8699.664} C_VEL
LIN {X 0,Y 359.421,Z 929.303,A -85,B 0,C 180,E1 -8702.549,E2 -8702.549} C_VEL
LIN {X 0,Y 357.001,Z 944.573,A -85,B 0,C 180,E1 -8705.687,E2 -8705.687} C_VEL
LIN {X 0,Y 355.1,Z 958.182,A -85,B 0,C 180,E1 -8709.047,E2 -8709.047} C_VEL
LIN {X 0,Y 353.813,Z 969.325,A -85,B 0,C 180,E1 -8712.399,E2 -8712.399} C_VEL
LIN {X 0,Y 353.063,Z 977.916,A -85,B 0,C 180,E1 -8715.586,E2 -8715.586} C_VEL
LIN {X 0,Y 352.702,Z 984.746,A -85,B 0,C 180,E1 -8718.77,E2 -8718.77} C_VEL
LIN {X 0,Y 352.563,Z 990.142,A -85,B 0,C 180,E1 -8722.176,E2 -8722.176} C_VEL
LIN {X 0,Y 352.572,Z 993.421,A -85,B 0,C 180,E1 -8725.282,E2 -8725.282} C_VEL
LIN {X 0,Y 352.594,Z 995.23,A -85,B 0,C 180,E1 -8728.537,E2 -8728.537} C_VEL
LIN {X 0,Y 352.575,Z 995.362,A -85,B 0,C 180,E1 -8731.625,E2 -8731.625} C_VEL
LIN {X 0,Y 352.497,Z 994.002,A -85,B 0,C 180,E1 -8734.718,E2 -8734.718} C_VEL
LIN {X 0,Y 352.452,Z 991.119,A -85,B 0,C 180,E1 -8737.826,E2 -8737.826} C_VEL
LIN {X 0,Y 352.557,Z 986.437,A -85,B 0,C 180,E1 -8741.119,E2 -8741.119} C_VEL
LIN {X 0,Y 352.937,Z 979.933,A -85,B 0,C 180,E1 -8744.436,E2 -8744.436} C_VEL
LIN {X 0,Y 353.71,Z 972.029,A -85,B 0,C 180,E1 -8747.605,E2 -8747.605} C_VEL
LIN {X 0,Y 355.067,Z 961.716,A -85,B 0,C 180,E1 -8750.954,E2 -8750.954} C_VEL
LIN {X 0,Y 356.955,Z 949.794,A -85,B 0,C 180,E1 -8754.139,E2 -8754.139} C_VEL
LIN {X 0,Y 359.523,Z 935.495,A -85,B 0,C 180,E1 -8757.314,E2 -8757.314} C_VEL
LIN {X 0,Y 362.648,Z 919.407,A -85,B 0,C 180,E1 -8760.301,E2 -8760.301} C_VEL
LIN {X 0,Y 366.042,Z 902.565,A -85,B 0,C 180,E1 -8762.927,E2 -8762.927} C_VEL
LIN {X 0,Y 369.745,Z 884.071,A -85,B 0,C 180,E1 -8765.358,E2 -8765.358} C_VEL
LIN {X 0,Y 373.407,Z 865.268,A -85,B 0,C 180,E1 -8767.432,E2 -8767.432} C_VEL
LIN {X 0,Y 377.213,Z 844.976,A -85,B 0,C 180,E1 -8769.309,E2 -8769.309} C_VEL
LIN {X 0,Y 380.771,Z 824.752,A -85,B 0,C 180,E1 -8770.866,E2 -8770.866} C_VEL
LIN {X 0,Y 384.113,Z 803.492,A -85,B 0,C 180,E1 -8772.189,E2 -8772.189} C_VEL
LIN {X 0,Y 387.159,Z 781.34,A -85,B 0,C 180,E1 -8773.278,E2 -8773.278} C_VEL
LIN {X 0,Y 389.808,Z 758.693,A -85,B 0,C 180,E1 -8774.116,E2 -8774.116} C_VEL
LIN {X 0,Y 391.577,Z 735.585,A -85,B 0,C 180,E1 -8774.744,E2 -8774.744} C_VEL
LIN {X 0,Y 393.165,Z 714.678,A -85,B 0,C 180,E1 -8775.163,E2 -8775.163} C_VEL
LIN {X 0,Y 394.057,Z 707.469,A -85,B 0,C 180,E1 -8775.272,E2 -8775.272} C_VEL
LIN {X 0,Y 404.13,Z 681.106,A -85,B 0,C 180,E1 -8776.564,E2 -8776.564} C_VEL
LIN {X 0,Y 412.559,Z 662.048,A -85,B 0,C 180,E1 -8777.353,E2 -8777.353} C_VEL
LIN {X 0,Y 420.344,Z 646.086,A -85,B 0,C 180,E1 -8777.914,E2 -8777.914} C_VEL
LIN {X 0,Y 430.5,Z 625.273,A -85,B 0,C 180,E1 -8778.606,E2 -8778.606} C_VEL
LIN {X 0,Y 431.97,Z 622.264,A -85,B 0,C 180,E1 -8778.703,E2 -8778.703} C_VEL
LIN {X 0,Y 424.592,Z 609.164,A -85,B 0,C 180,E1 -8780.695,E2 -8780.695} C_VEL
LIN {X 0,Y 418.383,Z 593.58,A -85,B 0,C 180,E1 -8782.885,E2 -8782.885} C_VEL
LIN {X 0,Y 414.33,Z 577.565,A -85,B 0,C 180,E1 -8784.947,E2 -8784.947} C_VEL
LIN {X 0,Y 411.981,Z 559.187,A -85,B 0,C 180,E1 -8787.111,E2 -8787.111} C_VEL
LIN {X 0,Y 411.608,Z 538.278,A -85,B 0,C 180,E1 -8789.328,E2 -8789.328} C_VEL
LIN {X 0,Y 413.358,Z 516.713,A -85,B 0,C 180,E1 -8791.385,E2 -8791.385} C_VEL
LIN {X 0,Y 416.246,Z 497.254,A -85,B 0,C 180,E1 -8793.07,E2 -8793.07} C_VEL
LIN {X 0,Y 407.08,Z 479.76,A -85,B 0,C 180,E1 -8796.707,E2 -8796.707} C_VEL
LIN {X 0,Y 398.761,Z 464.459,A -85,B 0,C 180,E1 -8800.215,E2 -8800.215} C_VEL
LIN {X 0,Y 391.389,Z 451.339,A -85,B 0,C 180,E1 -8803.527,E2 -8803.527} C_VEL
LIN {X 0,Y 385.481,Z 440.911,A -85,B 0,C 180,E1 -8806.348,E2 -8806.348} C_VEL
LIN {X 0,Y 380.014,Z 431.532,A -85,B 0,C 180,E1 -8809.08,E2 -8809.08} C_VEL
LIN {X 0,Y 374.764,Z 422.483,A -85,B 0,C 180,E1 -8811.871,E2 -8811.871} C_VEL
LIN {X 0,Y 371.79,Z 417.436,A -85,B 0,C 180,E1 -8813.515,E2 -8813.515} C_VEL
LIN {X 0,Y 368.904,Z 412.532,A -85,B 0,C 180,E1 -8815.181,E2 -8815.181} C_VEL
LIN {X 0,Y 365.793,Z 407.309,A -85,B 0,C 180,E1 -8817.023,E2 -8817.023} C_VEL
LIN {X 0,Y 363.034,Z 402.475,A -85,B 0,C 180,E1 -8818.738,E2 -8818.738} C_VEL
LIN {X 0,Y 360.689,Z 398.857,A -85,B 0,C 180,E1 -8820.159,E2 -8820.159} C_VEL
LIN {X 0,Y 359.757,Z 397.073,A -85,B 0,C 180,E1 -8820.797,E2 -8820.797} C_VEL
LIN {X 0,Y 357.446,Z 393.608,A -85,B 0,C 180,E1 -8822.245,E2 -8822.245} C_VEL
LIN {X 0,Y 356.592,Z 391.76,A -85,B 0,C 180,E1 -8822.893,E2 -8822.893} C_VEL
LIN {X 0,Y 354.479,Z 388.964,A -85,B 0,C 180,E1 -8824.206,E2 -8824.206} C_VEL
LIN {X 0,Y 353.868,Z 386.658,A -85,B 0,C 180,E1 -8824.944,E2 -8824.944} C_VEL
LIN {X 0,Y 353.854,Z 386.665,A -85,B 0,C 180,E1 -8829.105,E2 -8829.105} C_VEL
LIN {X 0,Y 353.873,Z 386.653,A -85,B 0,C 180,E1 -8833.397,E2 -8833.397} C_VEL
LIN {X 0,Y 353.853,Z 386.653,A -85,B 0,C 180,E1 -8837.599,E2 -8837.599} C_VEL
LIN {X 0,Y 353.877,Z 386.652,A -85,B 0,C 180,E1 -8841.724,E2 -8841.724} C_VEL
LIN {X 0,Y 353.85,Z 386.655,A -85,B 0,C 180,E1 -8845.975,E2 -8845.975} C_VEL
LIN {X 0,Y 353.881,Z 386.648,A -85,B 0,C 180,E1 -8850.166,E2 -8850.166} C_VEL
LIN {X 0,Y 353.848,Z 386.633,A -85,B 0,C 180,E1 -8854.412,E2 -8854.412} C_VEL
LIN {X 0,Y 353.877,Z 386.766,A -85,B 0,C 180,E1 -8857.433,E2 -8857.433} C_VEL
LIN {X 0,Y 354.849,Z 389.596,A -85,B 0,C 180,E1 -8857.912,E2 -8857.912} C_VEL
LIN {X 0,Y 356.845,Z 392.4,A -85,B 0,C 180,E1 -8858.58,E2 -8858.58} C_VEL
LIN {X 0,Y 358.647,Z 395.809,A -85,B 0,C 180,E1 -8859.261,E2 -8859.261} C_VEL
LIN {X 0,Y 364.529,Z 406.29,A -85,B 0,C 180,E1 -8861.379,E2 -8861.379} C_VEL
LIN {X 0,Y 372.059,Z 421.387,A -85,B 0,C 180,E1 -8864.11,E2 -8864.11} C_VEL
LIN {X 0,Y 379.825,Z 439.462,A -85,B 0,C 180,E1 -8867.039,E2 -8867.039} C_VEL
LIN {X 0,Y 385.713,Z 455.487,A -85,B 0,C 180,E1 -8869.361,E2 -8869.361} C_VEL
LIN {X 0,Y 383.41,Z 496.921,A -85,B 0,C 180,E1 -8872.642,E2 -8872.642} C_VEL
LIN {X 0,Y 383.358,Z 503.128,A -85,B 0,C 180,E1 -8873.066,E2 -8873.066} C_VEL
LIN {X 0,Y 384.108,Z 510.709,A -85,B 0,C 180,E1 -8873.329,E2 -8873.329} C_VEL
LIN {X 0,Y 377.972,Z 706.871,A -85,B 0,C 180,E1 -8877.155,E2 -8877.155} C_VEL
LIN {X 0,Y 377.339,Z 725.53,A -85,B 0,C 180,E1 -8877.745,E2 -8877.745} C_VEL
LIN {X 0,Y 376.241,Z 742.888,A -85,B 0,C 180,E1 -8878.546,E2 -8878.546} C_VEL
LIN {X 0,Y 374.612,Z 760.241,A -85,B 0,C 180,E1 -8879.617,E2 -8879.617} C_VEL
LIN {X 0,Y 372.564,Z 776.954,A -85,B 0,C 180,E1 -8880.939,E2 -8880.939} C_VEL
LIN {X 0,Y 370.28,Z 792.723,A -85,B 0,C 180,E1 -8882.5,E2 -8882.5} C_VEL
LIN {X 0,Y 367.768,Z 807.546,A -85,B 0,C 180,E1 -8884.302,E2 -8884.302} C_VEL
LIN {X 0,Y 365.071,Z 821.842,A -85,B 0,C 180,E1 -8886.431,E2 -8886.431} C_VEL
LIN {X 0,Y 362.612,Z 834.074,A -85,B 0,C 180,E1 -8888.656,E2 -8888.656} C_VEL
LIN {X 0,Y 360.236,Z 845.38,A -85,B 0,C 180,E1 -8891.169,E2 -8891.169} C_VEL
LIN {X 0,Y 358.236,Z 854.919,A -85,B 0,C 180,E1 -8893.794,E2 -8893.794} C_VEL
LIN {X 0,Y 356.616,Z 862.88,A -85,B 0,C 180,E1 -8896.544,E2 -8896.544} C_VEL
LIN {X 0,Y 355.36,Z 869.407,A -85,B 0,C 180,E1 -8899.462,E2 -8899.462} C_VEL
LIN {X 0,Y 354.51,Z 874.402,A -85,B 0,C 180,E1 -8902.546,E2 -8902.546} C_VEL
LIN {X 0,Y 354.076,Z 877.229,A -85,B 0,C 180,E1 -8905.207,E2 -8905.207} C_VEL
LIN {X 0,Y 352.975,Z 878.347,A -85,B 0,C 180,E1 -8906.438,E2 -8906.438} C_VEL
LIN {X 0,Y 348.266,Z 880.027,A -85,B 0,C 180,E1 -8908.772,E2 -8908.772} C_VEL
LIN {X 0,Y 346.092,Z 880.489,A -85,B 0,C 180,E1 -8910.299,E2 -8910.299} C_VEL
LIN {X 0,Y 345.893,Z 880.44,A -85,B 0,C 180,E1 -8910.852,E2 -8910.852} C_VEL
LIN {X 0,Y 346.073,Z 879.233,A -85,B 0,C 180,E1 -8913.977,E2 -8913.977} C_VEL
LIN {X 0,Y 346.536,Z 876.365,A -85,B 0,C 180,E1 -8917.127,E2 -8917.127} C_VEL
LIN {X 0,Y 347.312,Z 872.025,A -85,B 0,C 180,E1 -8920.115,E2 -8920.115} C_VEL
LIN {X 0,Y 348.532,Z 865.979,A -85,B 0,C 180,E1 -8923.099,E2 -8923.099} C_VEL
LIN {X 0,Y 350.138,Z 858.52,A -85,B 0,C 180,E1 -8925.911,E2 -8925.911} C_VEL
LIN {X 0,Y 352.221,Z 849.122,A -85,B 0,C 180,E1 -8928.71,E2 -8928.71} C_VEL
LIN {X 0,Y 354.671,Z 838.17,A -85,B 0,C 180,E1 -8931.326,E2 -8931.326} C_VEL
LIN {X 0,Y 357.37,Z 825.595,A -85,B 0,C 180,E1 -8933.759,E2 -8933.759} C_VEL
LIN {X 0,Y 360.061,Z 812.182,A -85,B 0,C 180,E1 -8935.878,E2 -8935.878} C_VEL
LIN {X 0,Y 362.725,Z 797.587,A -85,B 0,C 180,E1 -8937.767,E2 -8937.767} C_VEL
LIN {X 0,Y 365.226,Z 781.686,A -85,B 0,C 180,E1 -8939.443,E2 -8939.443} C_VEL
LIN {X 0,Y 367.329,Z 765.956,A -85,B 0,C 180,E1 -8940.78,E2 -8940.78} C_VEL
LIN {X 0,Y 369.15,Z 748.823,A -85,B 0,C 180,E1 -8941.928,E2 -8941.928} C_VEL
LIN {X 0,Y 370.498,Z 730.691,A -85,B 0,C 180,E1 -8942.845,E2 -8942.845} C_VEL
LIN {X 0,Y 371.271,Z 711.964,A -85,B 0,C 180,E1 -8943.505,E2 -8943.505} C_VEL
LIN {X 0,Y 372.471,Z 666.408,A -85,B 0,C 180,E1 -8944.469,E2 -8944.469} C_VEL
LIN {X 0,Y 377.723,Z 509.46,A -85,B 0,C 180,E1 -8947.559,E2 -8947.559} C_VEL
LIN {X 0,Y 376.972,Z 502.897,A -85,B 0,C 180,E1 -8947.833,E2 -8947.833} C_VEL
LIN {X 0,Y 379.06,Z 464.461,A -85,B 0,C 180,E1 -8950.856,E2 -8950.856} C_VEL
LIN {X 0,Y 379.379,Z 458.963,A -85,B 0,C 180,E1 -8951.312,E2 -8951.312} C_VEL
LIN {X 0,Y 374.436,Z 445.558,A -85,B 0,C 180,E1 -8953.309,E2 -8953.309} C_VEL
LIN {X 0,Y 372.998,Z 445.114,A -85,B 0,C 180,E1 -8953.598,E2 -8953.598} C_VEL
LIN {X 0,Y 379.413,Z 461.832,A -85,B 0,C 180,E1 -8956.664,E2 -8956.664} C_VEL
LIN {X 0,Y 380.825,Z 466.338,A -85,B 0,C 180,E1 -8957.411,E2 -8957.411} C_VEL
LIN {X 0,Y 375.396,Z 507.135,A -85,B 0,C 180,E1 -8961.543,E2 -8961.543} C_VEL
LIN {X 0,Y 370.094,Z 550.721,A -85,B 0,C 180,E1 -8965.903,E2 -8965.903} C_VEL
LIN {X 0,Y 365.002,Z 597.718,A -85,B 0,C 180,E1 -8970.556,E2 -8970.556} C_VEL
LIN {X 0,Y 363.946,Z 609.643,A -85,B 0,C 180,E1 -8971.688,E2 -8971.688} C_VEL
LIN {X 0,Y 364.534,Z 619.497,A -85,B 0,C 180,E1 -8972.067,E2 -8972.067} C_VEL
LIN {X 0,Y 357.326,Z 752.915,A -85,B 0,C 180,E1 -8976.024,E2 -8976.024} C_VEL
LIN {X 0,Y 356.58,Z 771.142,A -85,B 0,C 180,E1 -8976.798,E2 -8976.798} C_VEL
LIN {X 0,Y 355.569,Z 787.113,A -85,B 0,C 180,E1 -8977.776,E2 -8977.776} C_VEL
LIN {X 0,Y 354.355,Z 802.36,A -85,B 0,C 180,E1 -8979.001,E2 -8979.001} C_VEL
LIN {X 0,Y 352.908,Z 817.435,A -85,B 0,C 180,E1 -8980.555,E2 -8980.555} C_VEL
LIN {X 0,Y 351.5,Z 830.892,A -85,B 0,C 180,E1 -8982.279,E2 -8982.279} C_VEL
LIN {X 0,Y 350.103,Z 843.297,A -85,B 0,C 180,E1 -8984.257,E2 -8984.257} C_VEL
LIN {X 0,Y 348.886,Z 854.294,A -85,B 0,C 180,E1 -8986.408,E2 -8986.408} C_VEL
LIN {X 0,Y 347.811,Z 864.37,A -85,B 0,C 180,E1 -8988.895,E2 -8988.895} C_VEL
LIN {X 0,Y 347.071,Z 872.29,A -85,B 0,C 180,E1 -8991.384,E2 -8991.384} C_VEL
LIN {X 0,Y 346.607,Z 878.672,A -85,B 0,C 180,E1 -8994.039,E2 -8994.039} C_VEL
LIN {X 0,Y 346.441,Z 883.149,A -85,B 0,C 180,E1 -8996.69,E2 -8996.69} C_VEL
LIN {X 0,Y 346.531,Z 886.052,A -85,B 0,C 180,E1 -8999.504,E2 -8999.504} C_VEL
LIN {X 0,Y 346.855,Z 887.011,A -85,B 0,C 180,E1 -9002.147,E2 -9002.147} C_VEL
LIN {X 0,Y 347.502,Z 886.291,A -85,B 0,C 180,E1 -9004.951,E2 -9004.951} C_VEL
LIN {X 0,Y 348.505,Z 883.657,A -85,B 0,C 180,E1 -9007.749,E2 -9007.749} C_VEL
LIN {X 0,Y 349.86,Z 879.403,A -85,B 0,C 180,E1 -9010.372,E2 -9010.372} C_VEL
LIN {X 0,Y 351.661,Z 873.319,A -85,B 0,C 180,E1 -9012.98,E2 -9012.98} C_VEL
LIN {X 0,Y 353.887,Z 865.06,A -85,B 0,C 180,E1 -9015.569,E2 -9015.569} C_VEL
LIN {X 0,Y 356.262,Z 855.781,A -85,B 0,C 180,E1 -9017.813,E2 -9017.813} C_VEL
LIN {X 0,Y 358.825,Z 845.117,A -85,B 0,C 180,E1 -9019.873,E2 -9019.873} C_VEL
LIN {X 0,Y 361.712,Z 831.831,A -85,B 0,C 180,E1 -9021.911,E2 -9021.911} C_VEL
LIN {X 0,Y 364.421,Z 817.86,A -85,B 0,C 180,E1 -9023.614,E2 -9023.614} C_VEL
LIN {X 0,Y 366.968,Z 802.925,A -85,B 0,C 180,E1 -9025.067,E2 -9025.067} C_VEL
LIN {X 0,Y 369.485,Z 786.232,A -85,B 0,C 180,E1 -9026.346,E2 -9026.346} C_VEL
LIN {X 0,Y 374.457,Z 760.738,A -85,B 0,C 180,E1 -9028.03,E2 -9028.03} C_VEL
LIN {X 0,Y 383.172,Z 726.49,A -85,B 0,C 180,E1 -9029.98,E2 -9029.98} C_VEL
LIN {X 0,Y 392.834,Z 688.118,A -85,B 0,C 180,E1 -9031.836,E2 -9031.836} C_VEL
LIN {X 0,Y 400.004,Z 657.954,A -85,B 0,C 180,E1 -9033.104,E2 -9033.104} C_VEL
LIN {X 0,Y 407.644,Z 644.332,A -85,B 0,C 180,E1 -9033.96,E2 -9033.96} C_VEL
LIN {X 0,Y 418.322,Z 626.72,A -85,B 0,C 180,E1 -9036.353,E2 -9036.353} C_VEL
LIN {X 0,Y 426.31,Z 616.288,A -85,B 0,C 180,E1 -9037.829,E2 -9037.829} C_VEL
LIN {X 0,Y 426.286,Z 623.174,A -85,B 0,C 180,E1 -9039.706,E2 -9039.706} C_VEL
LIN {X 0,Y 426.992,Z 626.53,A -85,B 0,C 180,E1 -9040.573,E2 -9040.573} C_VEL
LIN {X 0,Y 416.88,Z 646.661,A -85,B 0,C 180,E1 -9041.243,E2 -9041.243} C_VEL
LIN {X 0,Y 403.673,Z 674.037,A -85,B 0,C 180,E1 -9042.217,E2 -9042.217} C_VEL
LIN {X 0,Y 398.693,Z 686.083,A -85,B 0,C 180,E1 -9042.755,E2 -9042.755} C_VEL
LIN {X 0,Y 391.263,Z 726.75,A -85,B 0,C 180,E1 -9043.635,E2 -9043.635} C_VEL
LIN {X 0,Y 386.465,Z 754.733,A -85,B 0,C 180,E1 -9044.702,E2 -9044.702} C_VEL
LIN {X 0,Y 381.069,Z 782.274,A -85,B 0,C 180,E1 -9046.052,E2 -9046.052} C_VEL
LIN {X 0,Y 376.233,Z 806.071,A -85,B 0,C 180,E1 -9047.544,E2 -9047.544} C_VEL
LIN {X 0,Y 371.017,Z 831.37,A -85,B 0,C 180,E1 -9049.497,E2 -9049.497} C_VEL
LIN {X 0,Y 366.328,Z 854.027,A -85,B 0,C 180,E1 -9051.615,E2 -9051.615} C_VEL
LIN {X 0,Y 361.752,Z 876.579,A -85,B 0,C 180,E1 -9054.129,E2 -9054.129} C_VEL
LIN {X 0,Y 357.626,Z 897.244,A -85,B 0,C 180,E1 -9056.866,E2 -9056.866} C_VEL
LIN {X 0,Y 354.026,Z 916.059,A -85,B 0,C 180,E1 -9059.82,E2 -9059.82} C_VEL
LIN {X 0,Y 351.054,Z 932.582,A -85,B 0,C 180,E1 -9062.889,E2 -9062.889} C_VEL
LIN {X 0,Y 348.62,Z 947.51,A -85,B 0,C 180,E1 -9066.191,E2 -9066.191} C_VEL
LIN {X 0,Y 346.855,Z 960.056,A -85,B 0,C 180,E1 -9069.529,E2 -9069.529} C_VEL
LIN {X 0,Y 345.689,Z 970.318,A -85,B 0,C 180,E1 -9072.841,E2 -9072.841} C_VEL
LIN {X 0,Y 345.005,Z 978.593,A -85,B 0,C 180,E1 -9076.133,E2 -9076.133} C_VEL
LIN {X 0,Y 344.697,Z 985.232,A -85,B 0,C 180,E1 -9079.522,E2 -9079.522} C_VEL
LIN {X 0,Y 344.615,Z 989.919,A -85,B 0,C 180,E1 -9082.833,E2 -9082.833} C_VEL
LIN {X 0,Y 344.666,Z 992.87,A -85,B 0,C 180,E1 -9086.007,E2 -9086.007} C_VEL
LIN {X 0,Y 344.674,Z 994.211,A -85,B 0,C 180,E1 -9089.168,E2 -9089.168} C_VEL
LIN {X 0,Y 344.638,Z 994.062,A -85,B 0,C 180,E1 -9092.327,E2 -9092.327} C_VEL
LIN {X 0,Y 344.558,Z 992.309,A -85,B 0,C 180,E1 -9095.54,E2 -9095.54} C_VEL
LIN {X 0,Y 344.513,Z 988.92,A -85,B 0,C 180,E1 -9098.848,E2 -9098.848} C_VEL
LIN {X 0,Y 344.676,Z 983.703,A -85,B 0,C 180,E1 -9102.225,E2 -9102.225} C_VEL
LIN {X 0,Y 345.16,Z 977.081,A -85,B 0,C 180,E1 -9105.456,E2 -9105.456} C_VEL
LIN {X 0,Y 346.148,Z 968.212,A -85,B 0,C 180,E1 -9108.875,E2 -9108.875} C_VEL
LIN {X 0,Y 347.756,Z 957.208,A -85,B 0,C 180,E1 -9112.304,E2 -9112.304} C_VEL
LIN {X 0,Y 349.956,Z 944.535,A -85,B 0,C 180,E1 -9115.557,E2 -9115.557} C_VEL
LIN {X 0,Y 352.888,Z 929.349,A -85,B 0,C 180,E1 -9118.794,E2 -9118.794} C_VEL
LIN {X 0,Y 356.301,Z 912.682,A -85,B 0,C 180,E1 -9121.758,E2 -9121.758} C_VEL
LIN {X 0,Y 359.897,Z 895.499,A -85,B 0,C 180,E1 -9124.33,E2 -9124.33} C_VEL
LIN {X 0,Y 363.674,Z 877.185,A -85,B 0,C 180,E1 -9126.627,E2 -9126.627} C_VEL
LIN {X 0,Y 367.623,Z 857.429,A -85,B 0,C 180,E1 -9128.722,E2 -9128.722} C_VEL
LIN {X 0,Y 371.52,Z 837.225,A -85,B 0,C 180,E1 -9130.511,E2 -9130.511} C_VEL
LIN {X 0,Y 375.084,Z 816.702,A -85,B 0,C 180,E1 -9131.996,E2 -9131.996} C_VEL
LIN {X 0,Y 378.624,Z 794.149,A -85,B 0,C 180,E1 -9133.309,E2 -9133.309} C_VEL
LIN {X 0,Y 381.669,Z 771.947,A -85,B 0,C 180,E1 -9134.311,E2 -9134.311} C_VEL
LIN {X 0,Y 384.123,Z 748.816,A -85,B 0,C 180,E1 -9135.086,E2 -9135.086} C_VEL
LIN {X 0,Y 386.325,Z 718.271,A -85,B 0,C 180,E1 -9135.8,E2 -9135.8} C_VEL
LIN {X 0,Y 387.822,Z 706.407,A -85,B 0,C 180,E1 -9135.996,E2 -9135.996} C_VEL
LIN {X 0,Y 398.804,Z 678.262,A -85,B 0,C 180,E1 -9137.378,E2 -9137.378} C_VEL
LIN {X 0,Y 407.869,Z 658.364,A -85,B 0,C 180,E1 -9138.178,E2 -9138.178} C_VEL
LIN {X 0,Y 414.97,Z 643.893,A -85,B 0,C 180,E1 -9138.686,E2 -9138.686} C_VEL
LIN {X 0,Y 424.299,Z 624.68,A -85,B 0,C 180,E1 -9139.349,E2 -9139.349} C_VEL
LIN {X 0,Y 416.689,Z 609.87,A -85,B 0,C 180,E1 -9141.576,E2 -9141.576} C_VEL
LIN {X 0,Y 411.074,Z 594.102,A -85,B 0,C 180,E1 -9143.769,E2 -9143.769} C_VEL
LIN {X 0,Y 407.334,Z 576.799,A -85,B 0,C 180,E1 -9145.968,E2 -9145.968} C_VEL
LIN {X 0,Y 405.565,Z 558.653,A -85,B 0,C 180,E1 -9148.075,E2 -9148.075} C_VEL
LIN {X 0,Y 405.729,Z 537.525,A -85,B 0,C 180,E1 -9150.309,E2 -9150.309} C_VEL
LIN {X 0,Y 407.99,Z 515.265,A -85,B 0,C 180,E1 -9152.408,E2 -9152.408} C_VEL
LIN {X 0,Y 410.139,Z 501.487,A -85,B 0,C 180,E1 -9153.618,E2 -9153.618} C_VEL
LIN {X 0,Y 401.727,Z 485.35,A -85,B 0,C 180,E1 -9156.999,E2 -9156.999} C_VEL
LIN {X 0,Y 392.845,Z 468.828,A -85,B 0,C 180,E1 -9160.833,E2 -9160.833} C_VEL
LIN {X 0,Y 384.006,Z 453.029,A -85,B 0,C 180,E1 -9164.908,E2 -9164.908} C_VEL
LIN {X 0,Y 376.485,Z 439.703,A -85,B 0,C 180,E1 -9168.667,E2 -9168.667} C_VEL
LIN {X 0,Y 369.448,Z 427.901,A -85,B 0,C 180,E1 -9172.38,E2 -9172.38} C_VEL
LIN {X 0,Y 366.719,Z 423.264,A -85,B 0,C 180,E1 -9173.896,E2 -9173.896} C_VEL
LIN {X 0,Y 364.072,Z 418.726,A -85,B 0,C 180,E1 -9175.432,E2 -9175.432} C_VEL
LIN {X 0,Y 360.947,Z 413.471,A -85,B 0,C 180,E1 -9177.301,E2 -9177.301} C_VEL
LIN {X 0,Y 357.909,Z 408.332,A -85,B 0,C 180,E1 -9179.2,E2 -9179.2} C_VEL
LIN {X 0,Y 355.009,Z 403.377,A -85,B 0,C 180,E1 -9181.067,E2 -9181.067} C_VEL
LIN {X 0,Y 352.615,Z 399.591,A -85,B 0,C 180,E1 -9182.601,E2 -9182.601} C_VEL
LIN {X 0,Y 351.975,Z 398.222,A -85,B 0,C 180,E1 -9183.094,E2 -9183.094} C_VEL
LIN {X 0,Y 349.625,Z 394.874,A -85,B 0,C 180,E1 -9184.593,E2 -9184.593} C_VEL
LIN {X 0,Y 348.891,Z 392.923,A -85,B 0,C 180,E1 -9185.262,E2 -9185.262} C_VEL
LIN {X 0,Y 346.712,Z 390.24,A -85,B 0,C 180,E1 -9186.624,E2 -9186.624} C_VEL
LIN {X 0,Y 345.937,Z 387.644,A -85,B 0,C 180,E1 -9187.535,E2 -9187.535} C_VEL
LIN {X 0,Y 345.906,Z 387.65,A -85,B 0,C 180,E1 -9191.843,E2 -9191.843} C_VEL
LIN {X 0,Y 345.926,Z 387.64,A -85,B 0,C 180,E1 -9195.938,E2 -9195.938} C_VEL
LIN {X 0,Y 345.915,Z 387.641,A -85,B 0,C 180,E1 -9200.472,E2 -9200.472} C_VEL
LIN {X 0,Y 345.905,Z 387.643,A -85,B 0,C 180,E1 -9204.423,E2 -9204.423} C_VEL
LIN {X 0,Y 345.929,Z 387.642,A -85,B 0,C 180,E1 -9208.863,E2 -9208.863} C_VEL
LIN {X 0,Y 345.891,Z 387.652,A -85,B 0,C 180,E1 -9213.117,E2 -9213.117} C_VEL
LIN {X 0,Y 345.934,Z 387.67,A -85,B 0,C 180,E1 -9215.862,E2 -9215.862} C_VEL
LIN {X 0,Y 346.995,Z 390.707,A -85,B 0,C 180,E1 -9216.412,E2 -9216.412} C_VEL
LIN {X 0,Y 348.985,Z 393.197,A -85,B 0,C 180,E1 -9217.092,E2 -9217.092} C_VEL
LIN {X 0,Y 350.979,Z 396.99,A -85,B 0,C 180,E1 -9217.898,E2 -9217.898} C_VEL
LIN {X 0,Y 356.921,Z 407.37,A -85,B 0,C 180,E1 -9220.115,E2 -9220.115} C_VEL
LIN {X 0,Y 364.304,Z 421.922,A -85,B 0,C 180,E1 -9222.895,E2 -9222.895} C_VEL
LIN {X 0,Y 371.826,Z 438.899,A -85,B 0,C 180,E1 -9225.778,E2 -9225.778} C_VEL
LIN {X 0,Y 378.188,Z 455.603,A -85,B 0,C 180,E1 -9228.321,E2 -9228.321} C_VEL
LIN {X 0,Y 379.329,Z 459.327,A -85,B 0,C 180,E1 -9228.83,E2 -9228.83} C_VEL
LIN {X 0,Y 376.983,Z 500.89,A -85,B 0,C 180,E1 -9232.121,E2 -9232.121} C_VEL
LIN {X 0,Y 377.067,Z 504.629,A -85,B 0,C 180,E1 -9232.352,E2 -9232.352} C_VEL
LIN {X 0,Y 377.753,Z 512.006,A -85,B 0,C 180,E1 -9232.611,E2 -9232.611} C_VEL
LIN {X 0,Y 371.347,Z 707.465,A -85,B 0,C 180,E1 -9236.475,E2 -9236.475} C_VEL
LIN {X 0,Y 370.693,Z 726.283,A -85,B 0,C 180,E1 -9237.073,E2 -9237.073} C_VEL
LIN {X 0,Y 369.507,Z 744.241,A -85,B 0,C 180,E1 -9237.913,E2 -9237.913} C_VEL
LIN {X 0,Y 367.815,Z 761.485,A -85,B 0,C 180,E1 -9238.994,E2 -9238.994} C_VEL
LIN {X 0,Y 365.677,Z 778.203,A -85,B 0,C 180,E1 -9240.337,E2 -9240.337} C_VEL
LIN {X 0,Y 363.288,Z 793.977,A -85,B 0,C 180,E1 -9241.925,E2 -9241.925} C_VEL
LIN {X 0,Y 360.606,Z 809.087,A -85,B 0,C 180,E1 -9243.796,E2 -9243.796} C_VEL
LIN {X 0,Y 357.834,Z 823.103,A -85,B 0,C 180,E1 -9245.924,E2 -9245.924} C_VEL
LIN {X 0,Y 355.145,Z 835.828,A -85,B 0,C 180,E1 -9248.291,E2 -9248.291} C_VEL
LIN {X 0,Y 352.705,Z 846.84,A -85,B 0,C 180,E1 -9250.802,E2 -9250.802} C_VEL
LIN {X 0,Y 350.633,Z 856.186,A -85,B 0,C 180,E1 -9253.432,E2 -9253.432} C_VEL
LIN {X 0,Y 348.886,Z 864.292,A -85,B 0,C 180,E1 -9256.297,E2 -9256.297} C_VEL
LIN {X 0,Y 347.519,Z 871.001,A -85,B 0,C 180,E1 -9259.39,E2 -9259.39} C_VEL
LIN {X 0,Y 346.626,Z 875.869,A -85,B 0,C 180,E1 -9262.542,E2 -9262.542} C_VEL
LIN {X 0,Y 346.123,Z 878.959,A -85,B 0,C 180,E1 -9265.693,E2 -9265.693} C_VEL
LIN {X 0,Y 345.901,Z 880.39,A -85,B 0,C 180,E1 -9268.841,E2 -9268.841} C_VEL
LIN {X 0,Y 345.893,Z 880.44,A -85,B 0,C 180,E1 -9270.852,E2 -9270.852} C_VEL
LIN {X 0,Y 344.948,Z 880.337,A -85,B 0,C 180,E1 -9272.131,E2 -9272.131} C_VEL
LIN {X 0,Y 340.278,Z 879.797,A -85,B 0,C 180,E1 -9274.734,E2 -9274.734} C_VEL
LIN {X 0,Y 338.625,Z 878.808,A -85,B 0,C 180,E1 -9276.207,E2 -9276.207} C_VEL
LIN {X 0,Y 338.564,Z 878.328,A -85,B 0,C 180,E1 -9276.672,E2 -9276.672} C_VEL
LIN {X 0,Y 339.351,Z 874.134,A -85,B 0,C 180,E1 -9279.84,E2 -9279.84} C_VEL
LIN {X 0,Y 340.577,Z 868.319,A -85,B 0,C 180,E1 -9282.919,E2 -9282.919} C_VEL
LIN {X 0,Y 342.296,Z 860.748,A -85,B 0,C 180,E1 -9285.937,E2 -9285.937} C_VEL
LIN {X 0,Y 344.512,Z 851.251,A -85,B 0,C 180,E1 -9288.89,E2 -9288.89} C_VEL
LIN {X 0,Y 346.949,Z 840.888,A -85,B 0,C 180,E1 -9291.469,E2 -9291.469} C_VEL
LIN {X 0,Y 349.733,Z 828.643,A -85,B 0,C 180,E1 -9293.952,E2 -9293.952} C_VEL
LIN {X 0,Y 352.584,Z 815.268,A -85,B 0,C 180,E1 -9296.166,E2 -9296.166} C_VEL
LIN {X 0,Y 355.511,Z 800.225,A -85,B 0,C 180,E1 -9298.197,E2 -9298.197} C_VEL
LIN {X 0,Y 358.104,Z 784.727,A -85,B 0,C 180,E1 -9299.894,E2 -9299.894} C_VEL
LIN {X 0,Y 360.435,Z 768.264,A -85,B 0,C 180,E1 -9301.342,E2 -9301.342} C_VEL
LIN {X 0,Y 362.399,Z 750.741,A -85,B 0,C 180,E1 -9302.548,E2 -9302.548} C_VEL
LIN {X 0,Y 363.835,Z 732.495,A -85,B 0,C 180,E1 -9303.495,E2 -9303.495} C_VEL
LIN {X 0,Y 364.662,Z 713.906,A -85,B 0,C 180,E1 -9304.17,E2 -9304.17} C_VEL
LIN {X 0,Y 365.766,Z 672.549,A -85,B 0,C 180,E1 -9305.073,E2 -9305.073} C_VEL
LIN {X 0,Y 371.436,Z 510.589,A -85,B 0,C 180,E1 -9308.308,E2 -9308.308} C_VEL
LIN {X 0,Y 370.715,Z 504.063,A -85,B 0,C 180,E1 -9308.588,E2 -9308.588} C_VEL
LIN {X 0,Y 373.101,Z 463.132,A -85,B 0,C 180,E1 -9311.84,E2 -9311.84} C_VEL
LIN {X 0,Y 370.214,Z 454.369,A -85,B 0,C 180,E1 -9313.102,E2 -9313.102} C_VEL
LIN {X 0,Y 369.43,Z 452.595,A -85,B 0,C 180,E1 -9313.39,E2 -9313.39} C_VEL
LIN {X 0,Y 367.875,Z 452.126,A -85,B 0,C 180,E1 -9313.699,E2 -9313.699} C_VEL
LIN {X 0,Y 374.248,Z 469.424,A -85,B 0,C 180,E1 -9316.859,E2 -9316.859} C_VEL
LIN {X 0,Y 368.755,Z 509.009,A -85,B 0,C 180,E1 -9320.919,E2 -9320.919} C_VEL
LIN {X 0,Y 363.186,Z 552.766,A -85,B 0,C 180,E1 -9325.354,E2 -9325.354} C_VEL
LIN {X 0,Y 357.956,Z 599.155,A -85,B 0,C 180,E1 -9330,E2 -9330} C_VEL
LIN {X 0,Y 356.906,Z 610.483,A -85,B 0,C 180,E1 -9331.09,E2 -9331.09} C_VEL
LIN {X 0,Y 357.463,Z 620.373,A -85,B 0,C 180,E1 -9331.482,E2 -9331.482} C_VEL
LIN {X 0,Y 349.908,Z 752.863,A -85,B 0,C 180,E1 -9335.533,E2 -9335.533} C_VEL
LIN {X 0,Y 349.126,Z 771.113,A -85,B 0,C 180,E1 -9336.317,E2 -9336.317} C_VEL
LIN {X 0,Y 348.03,Z 787.88,A -85,B 0,C 180,E1 -9337.358,E2 -9337.358} C_VEL
LIN {X 0,Y 346.686,Z 804.059,A -85,B 0,C 180,E1 -9338.691,E2 -9338.691} C_VEL
LIN {X 0,Y 345.177,Z 819.124,A -85,B 0,C 180,E1 -9340.292,E2 -9340.292} C_VEL
LIN {X 0,Y 343.666,Z 832.958,A -85,B 0,C 180,E1 -9342.125,E2 -9342.125} C_VEL
LIN {X 0,Y 342.187,Z 845.709,A -85,B 0,C 180,E1 -9344.232,E2 -9344.232} C_VEL
LIN {X 0,Y 340.95,Z 856.473,A -85,B 0,C 180,E1 -9346.431,E2 -9346.431} C_VEL
LIN {X 0,Y 339.871,Z 866.427,A -85,B 0,C 180,E1 -9348.975,E2 -9348.975} C_VEL
LIN {X 0,Y 339.131,Z 874.167,A -85,B 0,C 180,E1 -9351.522,E2 -9351.522} C_VEL
LIN {X 0,Y 338.684,Z 880.457,A -85,B 0,C 180,E1 -9354.239,E2 -9354.239} C_VEL
LIN {X 0,Y 338.539,Z 885.039,A -85,B 0,C 180,E1 -9357.122,E2 -9357.122} C_VEL
LIN {X 0,Y 338.684,Z 887.629,A -85,B 0,C 180,E1 -9359.83,E2 -9359.83} C_VEL
LIN {X 0,Y 339.094,Z 888.535,A -85,B 0,C 180,E1 -9362.704,E2 -9362.704} C_VEL
LIN {X 0,Y 339.802,Z 887.709,A -85,B 0,C 180,E1 -9365.402,E2 -9365.402} C_VEL
LIN {X 0,Y 340.937,Z 885.048,A -85,B 0,C 180,E1 -9368.262,E2 -9368.262} C_VEL
LIN {X 0,Y 342.45,Z 880.721,A -85,B 0,C 180,E1 -9370.94,E2 -9370.94} C_VEL
LIN {X 0,Y 344.417,Z 874.581,A -85,B 0,C 180,E1 -9373.6,E2 -9373.6} C_VEL
LIN {X 0,Y 346.874,Z 866.328,A -85,B 0,C 180,E1 -9376.236,E2 -9376.236} C_VEL
LIN {X 0,Y 349.671,Z 856.336,A -85,B 0,C 180,E1 -9378.678,E2 -9378.678} C_VEL
LIN {X 0,Y 352.706,Z 844.582,A -85,B 0,C 180,E1 -9380.927,E2 -9380.927} C_VEL
LIN {X 0,Y 355.892,Z 831.005,A -85,B 0,C 180,E1 -9382.986,E2 -9382.986} C_VEL
LIN {X 0,Y 359.169,Z 815.292,A -85,B 0,C 180,E1 -9384.857,E2 -9384.857} C_VEL
LIN {X 0,Y 362.21,Z 798.964,A -85,B 0,C 180,E1 -9386.386,E2 -9386.386} C_VEL
LIN {X 0,Y 367.014,Z 774.486,A -85,B 0,C 180,E1 -9388.207,E2 -9388.207} C_VEL
LIN {X 0,Y 374.553,Z 746.152,A -85,B 0,C 180,E1 -9390.034,E2 -9390.034} C_VEL
LIN {X 0,Y 385.647,Z 707.212,A -85,B 0,C 180,E1 -9392.106,E2 -9392.106} C_VEL
LIN {X 0,Y 394.852,Z 670.688,A -85,B 0,C 180,E1 -9393.723,E2 -9393.723} C_VEL
LIN {X 0,Y 397.466,Z 661.093,A -85,B 0,C 180,E1 -9394.123,E2 -9394.123} C_VEL
LIN {X 0,Y 405.206,Z 647.896,A -85,B 0,C 180,E1 -9394.922,E2 -9394.922} C_VEL
LIN {X 0,Y 417.056,Z 630.377,A -85,B 0,C 180,E1 -9397.34,E2 -9397.34} C_VEL
LIN {X 0,Y 421.618,Z 624.889,A -85,B 0,C 180,E1 -9398.153,E2 -9398.153} C_VEL
LIN {X 0,Y 421.679,Z 630.617,A -85,B 0,C 180,E1 -9399.696,E2 -9399.696} C_VEL
LIN {X 0,Y 408.658,Z 656.219,A -85,B 0,C 180,E1 -9400.562,E2 -9400.562} C_VEL
LIN {X 0,Y 398.613,Z 676.785,A -85,B 0,C 180,E1 -9401.33,E2 -9401.33} C_VEL
LIN {X 0,Y 395.982,Z 683.182,A -85,B 0,C 180,E1 -9401.606,E2 -9401.606} C_VEL
LIN {X 0,Y 392.912,Z 698.978,A -85,B 0,C 180,E1 -9401.986,E2 -9401.986} C_VEL
LIN {X 0,Y 387.409,Z 726.284,A -85,B 0,C 180,E1 -9402.591,E2 -9402.591} C_VEL
LIN {X 0,Y 382.191,Z 752.986,A -85,B 0,C 180,E1 -9403.64,E2 -9403.64} C_VEL
LIN {X 0,Y 376.249,Z 780.467,A -85,B 0,C 180,E1 -9405.018,E2 -9405.018} C_VEL
LIN {X 0,Y 370.582,Z 805.534,A -85,B 0,C 180,E1 -9406.633,E2 -9406.633} C_VEL
LIN {X 0,Y 365.04,Z 830.148,A -85,B 0,C 180,E1 -9408.587,E2 -9408.587} C_VEL
LIN {X 0,Y 359.682,Z 853.832,A -85,B 0,C 180,E1 -9410.874,E2 -9410.874} C_VEL
LIN {X 0,Y 354.797,Z 876.077,A -85,B 0,C 180,E1 -9413.432,E2 -9413.432} C_VEL
LIN {X 0,Y 350.443,Z 896.313,A -85,B 0,C 180,E1 -9416.195,E2 -9416.195} C_VEL
LIN {X 0,Y 346.726,Z 914.478,A -85,B 0,C 180,E1 -9419.115,E2 -9419.115} C_VEL
LIN {X 0,Y 343.554,Z 930.996,A -85,B 0,C 180,E1 -9422.247,E2 -9422.247} C_VEL
LIN {X 0,Y 340.98,Z 945.797,A -85,B 0,C 180,E1 -9425.577,E2 -9425.577} C_VEL
LIN {X 0,Y 339.033,Z 958.779,A -85,B 0,C 180,E1 -9429.093,E2 -9429.093} C_VEL
LIN {X 0,Y 337.755,Z 969.396,A -85,B 0,C 180,E1 -9432.602,E2 -9432.602} C_VEL
LIN {X 0,Y 337.056,Z 977.54,A -85,B 0,C 180,E1 -9435.935,E2 -9435.935} C_VEL
LIN {X 0,Y 336.748,Z 984.158,A -85,B 0,C 180,E1 -9439.392,E2 -9439.392} C_VEL
LIN {X 0,Y 336.678,Z 988.893,A -85,B 0,C 180,E1 -9442.834,E2 -9442.834} C_VEL
LIN {X 0,Y 336.746,Z 991.766,A -85,B 0,C 180,E1 -9446.058,E2 -9446.058} C_VEL
LIN {X 0,Y 336.757,Z 993.071,A -85,B 0,C 180,E1 -9449.319,E2 -9449.319} C_VEL
LIN {X 0,Y 336.717,Z 992.896,A -85,B 0,C 180,E1 -9452.382,E2 -9452.382} C_VEL
LIN {X 0,Y 336.63,Z 991.153,A -85,B 0,C 180,E1 -9455.624,E2 -9455.624} C_VEL
LIN {X 0,Y 336.57,Z 987.679,A -85,B 0,C 180,E1 -9459.058,E2 -9459.058} C_VEL
LIN {X 0,Y 336.742,Z 982.402,A -85,B 0,C 180,E1 -9462.518,E2 -9462.518} C_VEL
LIN {X 0,Y 337.264,Z 975.688,A -85,B 0,C 180,E1 -9465.827,E2 -9465.827} C_VEL
LIN {X 0,Y 338.246,Z 967.213,A -85,B 0,C 180,E1 -9469.154,E2 -9469.154} C_VEL
LIN {X 0,Y 339.929,Z 956.166,A -85,B 0,C 180,E1 -9472.663,E2 -9472.663} C_VEL
LIN {X 0,Y 342.232,Z 943.436,A -85,B 0,C 180,E1 -9475.991,E2 -9475.991} C_VEL
LIN {X 0,Y 345.119,Z 929.066,A -85,B 0,C 180,E1 -9479.125,E2 -9479.125} C_VEL
LIN {X 0,Y 348.737,Z 912.018,A -85,B 0,C 180,E1 -9482.227,E2 -9482.227} C_VEL
LIN {X 0,Y 352.698,Z 893.816,A -85,B 0,C 180,E1 -9484.988,E2 -9484.988} C_VEL
LIN {X 0,Y 356.553,Z 875.76,A -85,B 0,C 180,E1 -9487.28,E2 -9487.28} C_VEL
LIN {X 0,Y 360.849,Z 855.022,A -85,B 0,C 180,E1 -9489.487,E2 -9489.487} C_VEL
LIN {X 0,Y 364.733,Z 835.385,A -85,B 0,C 180,E1 -9491.232,E2 -9491.232} C_VEL
LIN {X 0,Y 368.629,Z 813.721,A -85,B 0,C 180,E1 -9492.8,E2 -9492.8} C_VEL
LIN {X 0,Y 372.099,Z 792.155,A -85,B 0,C 180,E1 -9494.049,E2 -9494.049} C_VEL
LIN {X 0,Y 375.251,Z 769.642,A -85,B 0,C 180,E1 -9495.063,E2 -9495.063} C_VEL
LIN {X 0,Y 377.744,Z 746.543,A -85,B 0,C 180,E1 -9495.84,E2 -9495.84} C_VEL
LIN {X 0,Y 379.876,Z 717.998,A -85,B 0,C 180,E1 -9496.507,E2 -9496.507} C_VEL
LIN {X 0,Y 381.482,Z 705.718,A -85,B 0,C 180,E1 -9496.717,E2 -9496.717} C_VEL
LIN {X 0,Y 392.777,Z 677.172,A -85,B 0,C 180,E1 -9498.124,E2 -9498.124} C_VEL
LIN {X 0,Y 402.342,Z 656.563,A -85,B 0,C 180,E1 -9498.957,E2 -9498.957} C_VEL
LIN {X 0,Y 409.266,Z 642.616,A -85,B 0,C 180,E1 -9499.445,E2 -9499.445} C_VEL
LIN {X 0,Y 416.771,Z 627.104,A -85,B 0,C 180,E1 -9499.988,E2 -9499.988} C_VEL
LIN {X 0,Y 409.219,Z 611.272,A -85,B 0,C 180,E1 -9502.351,E2 -9502.351} C_VEL
LIN {X 0,Y 403.952,Z 594.944,A -85,B 0,C 180,E1 -9504.607,E2 -9504.607} C_VEL
LIN {X 0,Y 400.623,Z 577.055,A -85,B 0,C 180,E1 -9506.868,E2 -9506.868} C_VEL
LIN {X 0,Y 399.305,Z 557.616,A -85,B 0,C 180,E1 -9509.115,E2 -9509.115} C_VEL
LIN {X 0,Y 399.968,Z 536.37,A -85,B 0,C 180,E1 -9511.335,E2 -9511.335} C_VEL
LIN {X 0,Y 402.749,Z 513.645,A -85,B 0,C 180,E1 -9513.458,E2 -9513.458} C_VEL
LIN {X 0,Y 403.979,Z 505.621,A -85,B 0,C 180,E1 -9514.177,E2 -9514.177} C_VEL
LIN {X 0,Y 395.729,Z 489.76,A -85,B 0,C 180,E1 -9517.573,E2 -9517.573} C_VEL
LIN {X 0,Y 387.175,Z 473.728,A -85,B 0,C 180,E1 -9521.324,E2 -9521.324} C_VEL
LIN {X 0,Y 378.639,Z 458.475,A -85,B 0,C 180,E1 -9525.315,E2 -9525.315} C_VEL
LIN {X 0,Y 371.408,Z 445.598,A -85,B 0,C 180,E1 -9528.981,E2 -9528.981} C_VEL
LIN {X 0,Y 364.615,Z 434.126,A -85,B 0,C 180,E1 -9532.595,E2 -9532.595} C_VEL
LIN {X 0,Y 361.659,Z 429.07,A -85,B 0,C 180,E1 -9534.289,E2 -9534.289} C_VEL
LIN {X 0,Y 358.963,Z 424.509,A -85,B 0,C 180,E1 -9535.847,E2 -9535.847} C_VEL
LIN {X 0,Y 356.082,Z 419.608,A -85,B 0,C 180,E1 -9537.586,E2 -9537.586} C_VEL
LIN {X 0,Y 353.001,Z 414.426,A -85,B 0,C 180,E1 -9539.514,E2 -9539.514} C_VEL
LIN {X 0,Y 350.311,Z 409.718,A -85,B 0,C 180,E1 -9541.309,E2 -9541.309} C_VEL
LIN {X 0,Y 347.797,Z 405.573,A -85,B 0,C 180,E1 -9542.967,E2 -9542.967} C_VEL
LIN {X 0,Y 344.789,Z 400.782,A -85,B 0,C 180,E1 -9544.991,E2 -9544.991} C_VEL
LIN {X 0,Y 344.224,Z 399.363,A -85,B 0,C 180,E1 -9545.501,E2 -9545.501} C_VEL
LIN {X 0,Y 341.84,Z 396.1,A -85,B 0,C 180,E1 -9547.057,E2 -9547.057} C_VEL
LIN {X 0,Y 341.106,Z 394.024,A -85,B 0,C 180,E1 -9547.801,E2 -9547.801} C_VEL
LIN {X 0,Y 338.717,Z 391.131,A -85,B 0,C 180,E1 -9549.344,E2 -9549.344} C_VEL
LIN {X 0,Y 337.951,Z 388.636,A -85,B 0,C 180,E1 -9550.312,E2 -9550.312} C_VEL
LIN {X 0,Y 337.991,Z 388.633,A -85,B 0,C 180,E1 -9554.564,E2 -9554.564} C_VEL
LIN {X 0,Y 337.963,Z 388.634,A -85,B 0,C 180,E1 -9558.992,E2 -9558.992} C_VEL
LIN {X 0,Y 337.974,Z 388.631,A -85,B 0,C 180,E1 -9563.171,E2 -9563.171} C_VEL
LIN {X 0,Y 337.994,Z 388.616,A -85,B 0,C 180,E1 -9567.675,E2 -9567.675} C_VEL
LIN {X 0,Y 337.977,Z 388.622,A -85,B 0,C 180,E1 -9571.892,E2 -9571.892} C_VEL
LIN {X 0,Y 338.002,Z 388.786,A -85,B 0,C 180,E1 -9574.198,E2 -9574.198} C_VEL
LIN {X 0,Y 339.3,Z 392.127,A -85,B 0,C 180,E1 -9574.868,E2 -9574.868} C_VEL
LIN {X 0,Y 341.1,Z 394.021,A -85,B 0,C 180,E1 -9575.479,E2 -9575.479} C_VEL
LIN {X 0,Y 342.946,Z 397.758,A -85,B 0,C 180,E1 -9576.289,E2 -9576.289} C_VEL
LIN {X 0,Y 344.246,Z 399.496,A -85,B 0,C 180,E1 -9576.751,E2 -9576.751} C_VEL
LIN {X 0,Y 352.232,Z 413.982,A -85,B 0,C 180,E1 -9579.907,E2 -9579.907} C_VEL
LIN {X 0,Y 359.135,Z 427.709,A -85,B 0,C 180,E1 -9582.574,E2 -9582.574} C_VEL
LIN {X 0,Y 366.437,Z 444.535,A -85,B 0,C 180,E1 -9585.473,E2 -9585.473} C_VEL
LIN {X 0,Y 372.619,Z 461.107,A -85,B 0,C 180,E1 -9588.012,E2 -9588.012} C_VEL
LIN {X 0,Y 373.058,Z 462.825,A -85,B 0,C 180,E1 -9588.24,E2 -9588.24} C_VEL
LIN {X 0,Y 370.643,Z 504.183,A -85,B 0,C 180,E1 -9591.525,E2 -9591.525} C_VEL
LIN {X 0,Y 371.468,Z 513.077,A -85,B 0,C 180,E1 -9591.865,E2 -9591.865} C_VEL
LIN {X 0,Y 364.774,Z 708.156,A -85,B 0,C 180,E1 -9595.774,E2 -9595.774} C_VEL
LIN {X 0,Y 364.087,Z 727.256,A -85,B 0,C 180,E1 -9596.385,E2 -9596.385} C_VEL
LIN {X 0,Y 362.82,Z 745.584,A -85,B 0,C 180,E1 -9597.256,E2 -9597.256} C_VEL
LIN {X 0,Y 361.063,Z 762.729,A -85,B 0,C 180,E1 -9598.348,E2 -9598.348} C_VEL
LIN {X 0,Y 358.832,Z 779.453,A -85,B 0,C 180,E1 -9599.713,E2 -9599.713} C_VEL
LIN {X 0,Y 356.334,Z 795.231,A -85,B 0,C 180,E1 -9601.327,E2 -9601.327} C_VEL
LIN {X 0,Y 353.618,Z 809.901,A -85,B 0,C 180,E1 -9603.168,E2 -9603.168} C_VEL
LIN {X 0,Y 350.834,Z 823.4,A -85,B 0,C 180,E1 -9605.233,E2 -9605.233} C_VEL
LIN {X 0,Y 347.911,Z 836.601,A -85,B 0,C 180,E1 -9607.707,E2 -9607.707} C_VEL
LIN {X 0,Y 345.385,Z 847.444,A -85,B 0,C 180,E1 -9610.202,E2 -9610.202} C_VEL
LIN {X 0,Y 343.165,Z 856.914,A -85,B 0,C 180,E1 -9612.886,E2 -9612.886} C_VEL
LIN {X 0,Y 341.316,Z 864.985,A -85,B 0,C 180,E1 -9615.755,E2 -9615.755} C_VEL
LIN {X 0,Y 339.861,Z 871.612,A -85,B 0,C 180,E1 -9618.804,E2 -9618.804} C_VEL
LIN {X 0,Y 338.898,Z 876.465,A -85,B 0,C 180,E1 -9621.859,E2 -9621.859} C_VEL
LIN {X 0,Y 338.309,Z 879.846,A -85,B 0,C 180,E1 -9625.084,E2 -9625.084} C_VEL
LIN {X 0,Y 338.027,Z 881.549,A -85,B 0,C 180,E1 -9628.305,E2 -9628.305} C_VEL
LIN {X 0,Y 338.015,Z 881.626,A -85,B 0,C 180,E1 -9631.526,E2 -9631.526} C_VEL
LIN {X 0,Y 338.279,Z 880.076,A -85,B 0,C 180,E1 -9634.748,E2 -9634.748} C_VEL
LIN {X 0,Y 338.564,Z 878.328,A -85,B 0,C 180,E1 -9636.672,E2 -9636.672} C_VEL
LIN {X 0,Y 337.845,Z 877.049,A -85,B 0,C 180,E1 -9637.961,E2 -9637.961} C_VEL
LIN {X 0,Y 332.856,Z 873.135,A -85,B 0,C 180,E1 -9641.331,E2 -9641.331} C_VEL
LIN {X 0,Y 332.526,Z 871.056,A -85,B 0,C 180,E1 -9642.525,E2 -9642.525} C_VEL
LIN {X 0,Y 334.237,Z 863.927,A -85,B 0,C 180,E1 -9645.619,E2 -9645.619} C_VEL
LIN {X 0,Y 336.368,Z 855.236,A -85,B 0,C 180,E1 -9648.546,E2 -9648.546} C_VEL
LIN {X 0,Y 338.886,Z 845.062,A -85,B 0,C 180,E1 -9651.279,E2 -9651.279} C_VEL
LIN {X 0,Y 341.695,Z 833.416,A -85,B 0,C 180,E1 -9653.817,E2 -9653.817} C_VEL
LIN {X 0,Y 344.692,Z 820.22,A -85,B 0,C 180,E1 -9656.163,E2 -9656.163} C_VEL
LIN {X 0,Y 347.67,Z 805.94,A -85,B 0,C 180,E1 -9658.235,E2 -9658.235} C_VEL
LIN {X 0,Y 350.474,Z 790.65,A -85,B 0,C 180,E1 -9660.046,E2 -9660.046} C_VEL
LIN {X 0,Y 353.01,Z 774.375,A -85,B 0,C 180,E1 -9661.601,E2 -9661.601} C_VEL
LIN {X 0,Y 355.212,Z 757.046,A -85,B 0,C 180,E1 -9662.906,E2 -9662.906} C_VEL
LIN {X 0,Y 356.891,Z 738.841,A -85,B 0,C 180,E1 -9663.954,E2 -9663.954} C_VEL
LIN {X 0,Y 357.953,Z 720.408,A -85,B 0,C 180,E1 -9664.714,E2 -9664.714} C_VEL
LIN {X 0,Y 358.5,Z 697.839,A -85,B 0,C 180,E1 -9665.303,E2 -9665.303} C_VEL
LIN {X 0,Y 365.229,Z 511.84,A -85,B 0,C 180,E1 -9669.077,E2 -9669.077} C_VEL
LIN {X 0,Y 364.524,Z 505.235,A -85,B 0,C 180,E1 -9669.369,E2 -9669.369} C_VEL
LIN {X 0,Y 366.883,Z 466.005,A -85,B 0,C 180,E1 -9672.507,E2 -9672.507} C_VEL
LIN {X 0,Y 364.463,Z 459.765,A -85,B 0,C 180,E1 -9673.479,E2 -9673.479} C_VEL
LIN {X 0,Y 362.704,Z 459.301,A -85,B 0,C 180,E1 -9673.833,E2 -9673.833} C_VEL
LIN {X 0,Y 367.649,Z 472.864,A -85,B 0,C 180,E1 -9676.338,E2 -9676.338} C_VEL
LIN {X 0,Y 361.687,Z 514.244,A -85,B 0,C 180,E1 -9680.621,E2 -9680.621} C_VEL
LIN {X 0,Y 355.795,Z 559.095,A -85,B 0,C 180,E1 -9685.216,E2 -9685.216} C_VEL
LIN {X 0,Y 350.458,Z 604.893,A -85,B 0,C 180,E1 -9689.859,E2 -9689.859} C_VEL
LIN {X 0,Y 349.9,Z 611.372,A -85,B 0,C 180,E1 -9690.472,E2 -9690.472} C_VEL
LIN {X 0,Y 350.41,Z 621.315,A -85,B 0,C 180,E1 -9690.879,E2 -9690.879} C_VEL
LIN {X 0,Y 342.494,Z 752.554,A -85,B 0,C 180,E1 -9695.025,E2 -9695.025} C_VEL
LIN {X 0,Y 341.719,Z 770.433,A -85,B 0,C 180,E1 -9695.789,E2 -9695.789} C_VEL
LIN {X 0,Y 340.602,Z 787.475,A -85,B 0,C 180,E1 -9696.835,E2 -9696.835} C_VEL
LIN {X 0,Y 339.169,Z 804.174,A -85,B 0,C 180,E1 -9698.221,E2 -9698.221} C_VEL
LIN {X 0,Y 337.712,Z 818.458,A -85,B 0,C 180,E1 -9699.732,E2 -9699.732} C_VEL
LIN {X 0,Y 336.108,Z 832.724,A -85,B 0,C 180,E1 -9701.619,E2 -9701.619} C_VEL
LIN {X 0,Y 334.596,Z 845.266,A -85,B 0,C 180,E1 -9703.686,E2 -9703.686} C_VEL
LIN {X 0,Y 333.274,Z 856.371,A -85,B 0,C 180,E1 -9705.935,E2 -9705.935} C_VEL
LIN {X 0,Y 332.175,Z 865.982,A -85,B 0,C 180,E1 -9708.365,E2 -9708.365} C_VEL
LIN {X 0,Y 331.353,Z 874.206,A -85,B 0,C 180,E1 -9710.972,E2 -9710.972} C_VEL
LIN {X 0,Y 330.833,Z 880.825,A -85,B 0,C 180,E1 -9713.753,E2 -9713.753} C_VEL
LIN {X 0,Y 330.655,Z 885.604,A -85,B 0,C 180,E1 -9716.532,E2 -9716.532} C_VEL
LIN {X 0,Y 330.758,Z 888.733,A -85,B 0,C 180,E1 -9719.48,E2 -9719.48} C_VEL
LIN {X 0,Y 331.147,Z 890.001,A -85,B 0,C 180,E1 -9722.249,E2 -9722.249} C_VEL
LIN {X 0,Y 331.957,Z 889.478,A -85,B 0,C 180,E1 -9725.357,E2 -9725.357} C_VEL
LIN {X 0,Y 333.14,Z 887.053,A -85,B 0,C 180,E1 -9728.283,E2 -9728.283} C_VEL
LIN {X 0,Y 334.737,Z 883.052,A -85,B 0,C 180,E1 -9731.02,E2 -9731.02} C_VEL
LIN {X 0,Y 336.955,Z 876.82,A -85,B 0,C 180,E1 -9733.907,E2 -9733.907} C_VEL
LIN {X 0,Y 339.57,Z 868.836,A -85,B 0,C 180,E1 -9736.595,E2 -9736.595} C_VEL
LIN {X 0,Y 342.535,Z 859.162,A -85,B 0,C 180,E1 -9739.082,E2 -9739.082} C_VEL
LIN {X 0,Y 345.506,Z 848.738,A -85,B 0,C 180,E1 -9741.206,E2 -9741.206} C_VEL
LIN {X 0,Y 348.606,Z 837.098,A -85,B 0,C 180,E1 -9743.137,E2 -9743.137} C_VEL
LIN {X 0,Y 351.906,Z 823.537,A -85,B 0,C 180,E1 -9744.956,E2 -9744.956} C_VEL
LIN {X 0,Y 355.238,Z 808.435,A -85,B 0,C 180,E1 -9746.584,E2 -9746.584} C_VEL
LIN {X 0,Y 359.096,Z 790.099,A -85,B 0,C 180,E1 -9748.161,E2 -9748.161} C_VEL
LIN {X 0,Y 365.816,Z 765.034,A -85,B 0,C 180,E1 -9750.011,E2 -9750.011} C_VEL
LIN {X 0,Y 375.21,Z 735.241,A -85,B 0,C 180,E1 -9751.845,E2 -9751.845} C_VEL
LIN {X 0,Y 385.299,Z 701.82,A -85,B 0,C 180,E1 -9753.555,E2 -9753.555} C_VEL
LIN {X 0,Y 395.159,Z 664.712,A -85,B 0,C 180,E1 -9755.144,E2 -9755.144} C_VEL
LIN {X 0,Y 403.216,Z 651.59,A -85,B 0,C 180,E1 -9755.905,E2 -9755.905} C_VEL
LIN {X 0,Y 415.508,Z 635.115,A -85,B 0,C 180,E1 -9758.201,E2 -9758.201} C_VEL
LIN {X 0,Y 417.077,Z 633.384,A -85,B 0,C 180,E1 -9758.469,E2 -9758.469} C_VEL
LIN {X 0,Y 416.991,Z 634.568,A -85,B 0,C 180,E1 -9758.78,E2 -9758.78} C_VEL
LIN {X 0,Y 405.683,Z 656.269,A -85,B 0,C 180,E1 -9759.517,E2 -9759.517} C_VEL
LIN {X 0,Y 395.19,Z 677.036,A -85,B 0,C 180,E1 -9760.286,E2 -9760.286} C_VEL
LIN {X 0,Y 393.861,Z 680.751,A -85,B 0,C 180,E1 -9760.425,E2 -9760.425} C_VEL
LIN {X 0,Y 390.606,Z 696.262,A -85,B 0,C 180,E1 -9760.837,E2 -9760.837} C_VEL
LIN {X 0,Y 384.058,Z 725.836,A -85,B 0,C 180,E1 -9761.498,E2 -9761.498} C_VEL
LIN {X 0,Y 378.177,Z 752.224,A -85,B 0,C 180,E1 -9762.564,E2 -9762.564} C_VEL
LIN {X 0,Y 371.789,Z 778.838,A -85,B 0,C 180,E1 -9763.935,E2 -9763.935} C_VEL
LIN {X 0,Y 365.577,Z 803.642,A -85,B 0,C 180,E1 -9765.559,E2 -9765.559} C_VEL
LIN {X 0,Y 359.644,Z 827.632,A -85,B 0,C 180,E1 -9767.501,E2 -9767.501} C_VEL
LIN {X 0,Y 353.679,Z 851.72,A -85,B 0,C 180,E1 -9769.867,E2 -9769.867} C_VEL
LIN {X 0,Y 348.441,Z 873.581,A -85,B 0,C 180,E1 -9772.426,E2 -9772.426} C_VEL
LIN {X 0,Y 343.732,Z 893.876,A -85,B 0,C 180,E1 -9775.24,E2 -9775.24} C_VEL
LIN {X 0,Y 339.573,Z 912.658,A -85,B 0,C 180,E1 -9778.314,E2 -9778.314} C_VEL
LIN {X 0,Y 336.098,Z 929.512,A -85,B 0,C 180,E1 -9781.576,E2 -9781.576} C_VEL
